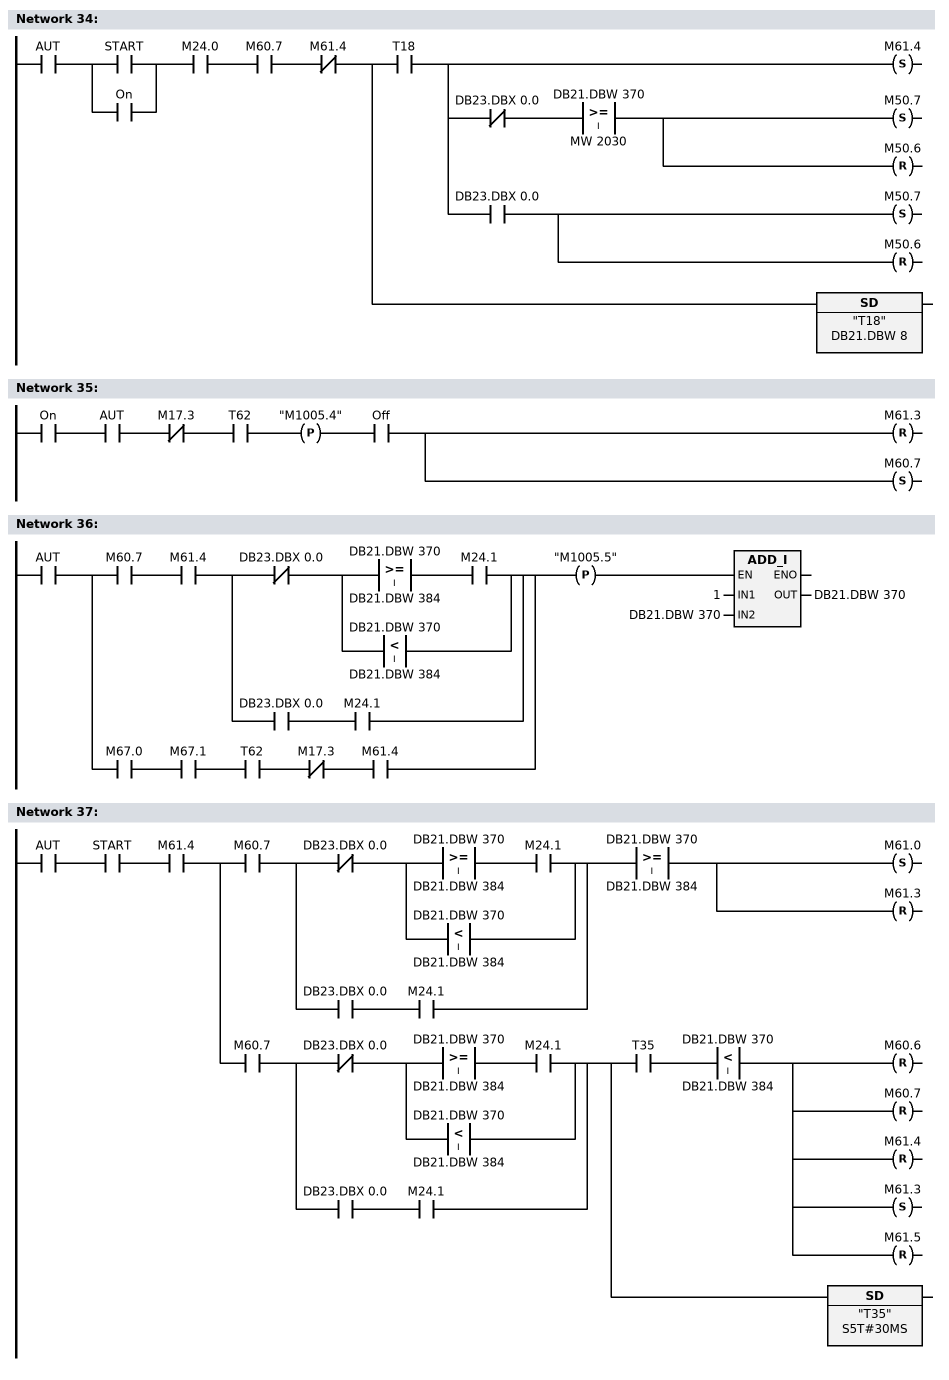
[picture p24: FC14 - AUTOMATIC networks 34-37]
NETWORK
TITLE =
      A     "AUT";
      A(;
      O     "START";
      O     "On";
      );
      A     "M24.0";
      A     "M60.7";
      AN    "M61.4";
      =     L 24.0;
      A     L 24.0;
      A     "T18";
      =     L 24.1;
      A     L 24.1;
      BLD   102;
      S     "M61.4";
      A     L 24.1;
      AN    DB23.DBX 0.0;
      A(;
      L     DB21.DBW 370;
      L     MW 2030;
      >=I;
      );
      S     "M50.7";
      R     "M50.6";
      A     L 24.1;
      A     DB23.DBX 0.0;
      S     "M50.7";
      R     "M50.6";
      A     L 24.0;
      BLD   102;
      L     DB21.DBW 8;
      SD    "T18";
NETWORK
TITLE =
      A     "On";
      A     "AUT";
      AN    "M17.3";
      A     "T62";
      FP    "M1005.4";
      A     "Off";
      R     "M61.3";
      S     "M60.7";
NETWORK
TITLE =
      A     "AUT";
      A(;
      A     "M60.7";
      A     "M61.4";
      A(;
      AN    DB23.DBX 0.0;
      A(;
      A(;
      L     DB21.DBW 370;
      L     DB21.DBW 384;
      >=I;
      );
      A     "M24.1";
      O(;
      L     DB21.DBW 370;
      L     DB21.DBW 384;
      <I;
      );
      );
      O;
      A     DB23.DBX 0.0;
      A     "M24.1";
      );
      O;
      A     "M67.0";
      A     "M67.1";
      A     "T62";
      AN    "M17.3";
      A     "M61.4";
      );
      FP    "M1005.5";
      JNB   M025;
      L     1;
      L     DB21.DBW 370;
      +I;
      T     DB21.DBW 370;
M025: NOP   0;
NETWORK
TITLE =
      A     "AUT";
      A     "START";
      A     "M61.4";
      =     L 24.0;
      A     L 24.0;
      A     "M60.7";
      A(;
      AN    DB23.DBX 0.0;
      A(;
      A(;
      L     DB21.DBW 370;
      L     DB21.DBW 384;
      >=I;
      );
      A     "M24.1";
      O(;
      L     DB21.DBW 370;
      L     DB21.DBW 384;
      <I;
      );
      );
      O;
      A     DB23.DBX 0.0;
      A     "M24.1";
      );
      A(;
      L     DB21.DBW 370;
      L     DB21.DBW 384;
      >=I;
      );
      S     "M61.0";
      R     "M61.3";
      A     L 24.0;
      A     "M60.7";
      A(;
      AN    DB23.DBX 0.0;
      A(;
      A(;
      L     DB21.DBW 370;
      L     DB21.DBW 384;
      >=I;
      );
      A     "M24.1";
      O(;
      L     DB21.DBW 370;
      L     DB21.DBW 384;
      <I;
      );
      );
      O;
      A     DB23.DBX 0.0;
      A     "M24.1";
      );
      =     L 24.1;
      A     L 24.1;
      A     "T35";
      A(;
      L     DB21.DBW 370;
      L     DB21.DBW 384;
      <I;
      );
      R     "M60.6";
      R     "M60.7";
      R     "M61.4";
      S     "M61.3";
      R     "M61.5";
      A     L 24.1;
      BLD   102;
      L     S5T#30MS;
      SD    "T35";
NETWORK
TITLE =
NETWORK
TITLE =
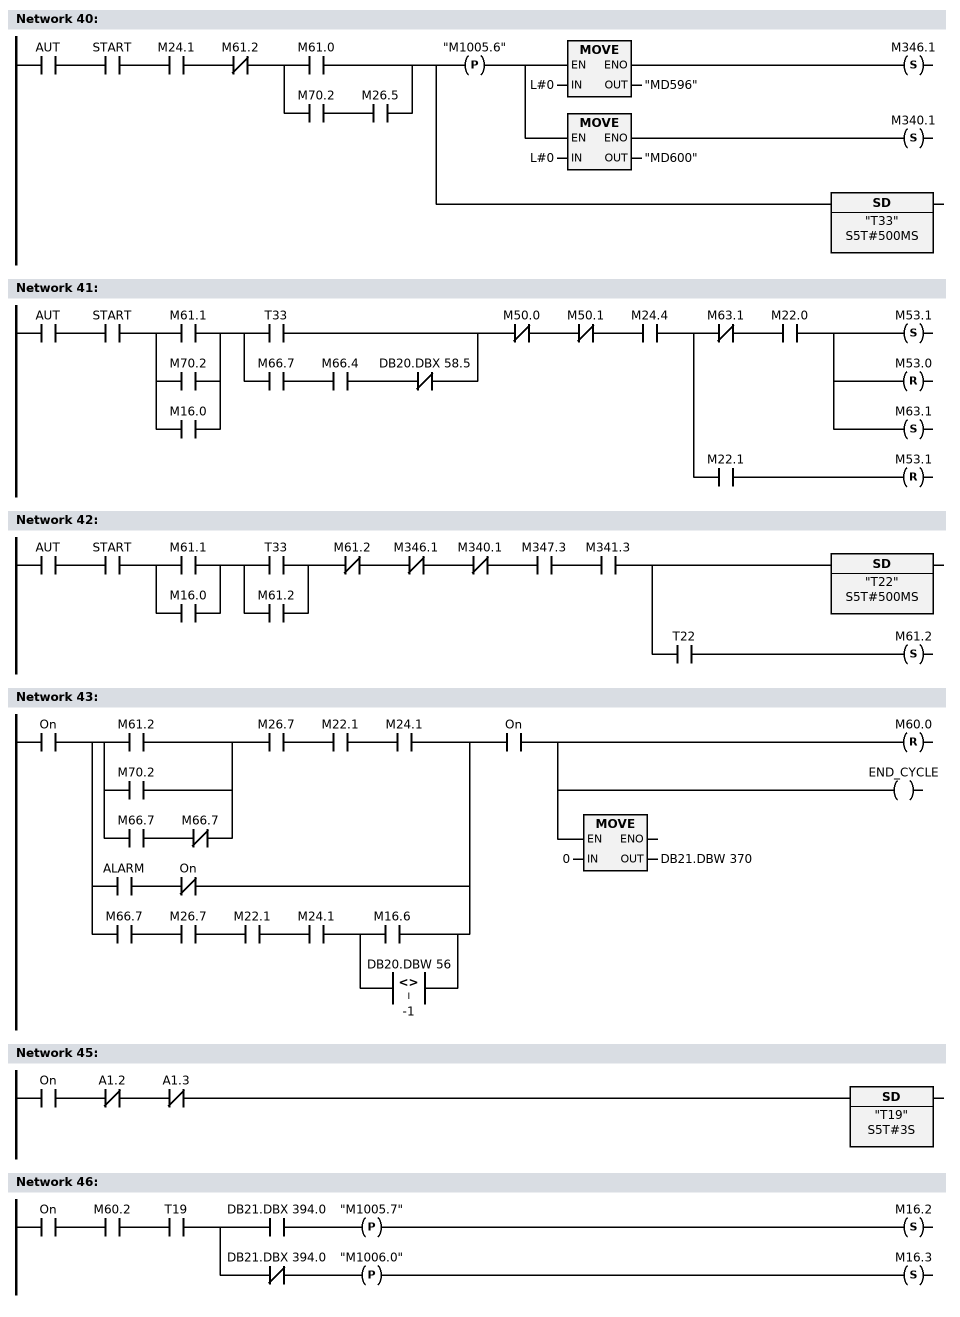
NETWORK
TITLE =
      A     "AUT";
      A     "START";
      A     "M24.1";
      AN    "M61.2";
      A(;
      O     "M61.0";
      O;
      A     "M70.2";
      A     "M26.5";
      );
      =     L 24.0;
      A     L 24.0;
      FP    "M1005.6";
      =     L 24.1;
      A     L 24.1;
      JNB   M026;
      L     L#0;
      T     "MD596";
      SET;
      SAVE;
      CLR;
M026: A     BR;
      S     "M346.1";
      A     L 24.1;
      JNB   M027;
      L     L#0;
      T     "MD600";
      SET;
      SAVE;
      CLR;
M027: A     BR;
      S     "M340.1";
      A     L 24.0;
      BLD   102;
      L     S5T#500MS;
      SD    "T33";
NETWORK
TITLE =
      A     "AUT";
      A     "START";
      A(;
      O     "M61.1";
      O     "M70.2";
      O     "M16.0";
      );
      A(;
      O     "T33";
      O;
      A     "M66.7";
      A     "M66.4";
      AN    DB20.DBX 58.5;
      );
      AN    "M50.0";
      AN    "M50.1";
      A     "M24.4";
      =     L 24.0;
      A     L 24.0;
      AN    "M63.1";
      A     "M22.0";
      S     "M53.1";
      R     "M53.0";
      S     "M63.1";
      A     L 24.0;
      A     "M22.1";
      R     "M53.1";
NETWORK
TITLE =
      A     "AUT";
      A     "START";
      A(;
      O     "M61.1";
      O     "M16.0";
      );
      A(;
      O     "T33";
      O     "M61.2";
      );
      AN    "M61.2";
      AN    "M346.1";
      AN    "M340.1";
      A     "M347.3";
      A     "M341.3";
      =     L 24.0;
      A     L 24.0;
      BLD   102;
      L     S5T#500MS;
      SD    "T22";
      A     L 24.0;
      A     "T22";
      S     "M61.2";
NETWORK
TITLE =
      A     "On";
      A(;
      A(;
      O     "M61.2";
      O     "M70.2";
      O;
      A     "M66.7";
      AN    "M66.7";
      );
      A     "M26.7";
      A     "M22.1";
      A     "M24.1";
      O;
      A     "ALARM";
      AN    "On";
      O;
      A     "M66.7";
      A     "M26.7";
      A     "M22.1";
      A     "M24.1";
      A(;
      O     "M16.6";
      O(;
      L     DB20.DBW 56;
      L     -1;
      <>I;
      );
      );
      );
      A     "On";
      =     L 24.0;
      A     L 24.0;
      BLD   102;
      R     "M60.0";
      A     L 24.0;
      BLD   102;
      =     "END_CYCLE";
      A     L 24.0;
      JNB   M028;
      L     0;
      T     DB21.DBW 370;
M028: NOP   0;
NETWORK
TITLE =
NETWORK
TITLE =
      A     "On";
      AN    "A1.2";
      AN    "A1.3";
      L     S5T#3S;
      SD    "T19";
NETWORK
TITLE =
      A     "On";
      A     "M60.2";
      A     "T19";
      =     L 24.0;
      A     L 24.0;
      A     DB21.DBX 394.0;
      FP    "M1005.7";
      S     "M16.2";
      A     L 24.0;
      AN    DB21.DBX 394.0;
      FP    "M1006.0";
      S     "M16.3";
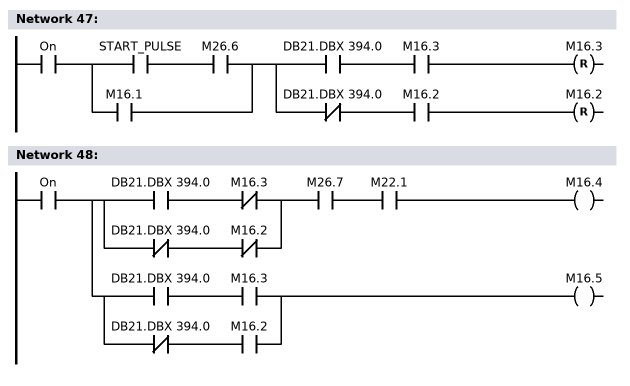
NETWORK
TITLE =
      A     "On";
      A(;
      A     "START_PULSE";
      A     "M26.6";
      O     "M16.1";
      );
      =     L 24.0;
      A     L 24.0;
      A     DB21.DBX 394.0;
      A     "M16.3";
      R     "M16.3";
      A     L 24.0;
      AN    DB21.DBX 394.0;
      A     "M16.2";
      R     "M16.2";
NETWORK
TITLE =
      A     "On";
      =     L 24.0;
      A     L 24.0;
      A(;
      A     DB21.DBX 394.0;
      AN    "M16.3";
      O;
      AN    DB21.DBX 394.0;
      AN    "M16.2";
      );
      A     "M26.7";
      A     "M22.1";
      =     "M16.4";
      A     L 24.0;
      A(;
      A     DB21.DBX 394.0;
      A     "M16.3";
      O;
      AN    DB21.DBX 394.0;
      A     "M16.2";
      );
      =     "M16.5";
END_FUNCTION

FUNCTION "FC16 - ALARMS" : VOID	// FC 16
VERSION : 0.1
BEGIN
// (block stored without names or comments; labels and parameter names are numbered)
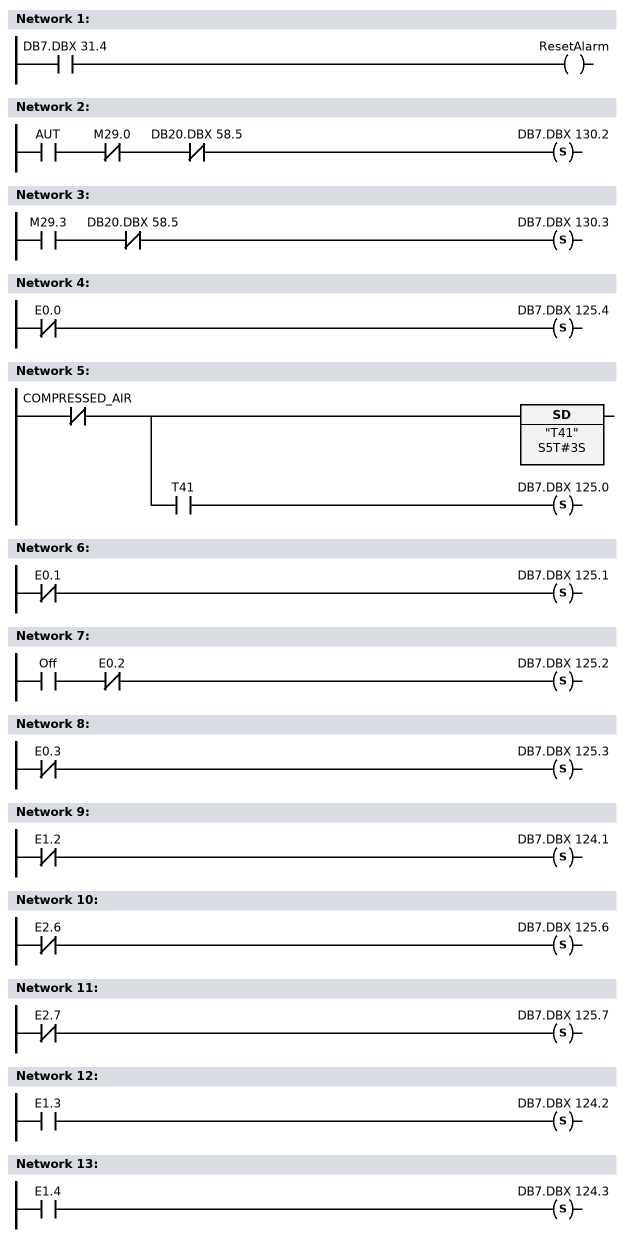
NETWORK
TITLE =
      A     DB7.DBX 31.4;
      =     "ResetAlarm";
NETWORK
TITLE =
      A     "AUT";
      AN    "M29.0";
      AN    DB20.DBX 58.5;
      S     DB7.DBX 130.2;
NETWORK
TITLE =
      A     "M29.3";
      AN    DB20.DBX 58.5;
      S     DB7.DBX 130.3;
NETWORK
TITLE =
      AN    "E0.0";
      S     DB7.DBX 125.4;
NETWORK
TITLE =
      AN    "COMPRESSED_AIR";
      =     L 1.0;
      A     L 1.0;
      BLD   102;
      L     S5T#3S;
      SD    "T41";
      A     L 1.0;
      A     "T41";
      S     DB7.DBX 125.0;
NETWORK
TITLE =
      AN    "E0.1";
      S     DB7.DBX 125.1;
NETWORK
TITLE =
      A     "Off";
      AN    "E0.2";
      S     DB7.DBX 125.2;
NETWORK
TITLE =
      AN    "E0.3";
      S     DB7.DBX 125.3;
NETWORK
TITLE =
      AN    "E1.2";
      S     DB7.DBX 124.1;
NETWORK
TITLE =
      AN    "E2.6";
      S     DB7.DBX 125.6;
NETWORK
TITLE =
      AN    "E2.7";
      S     DB7.DBX 125.7;
NETWORK
TITLE =
      A     "E1.3";
      S     DB7.DBX 124.2;
NETWORK
TITLE =
      A     "E1.4";
      S     DB7.DBX 124.3;
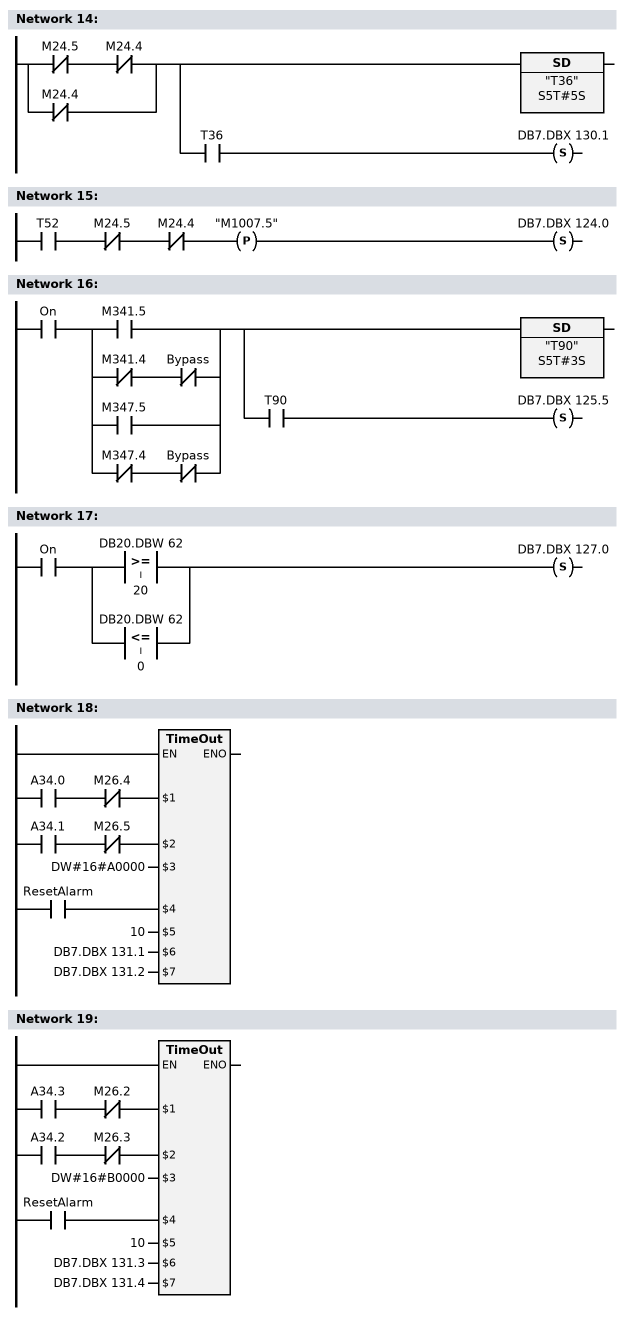
NETWORK
TITLE =
      AN    "M24.5";
      AN    "M24.4";
      ON    "M24.4";
      =     L 1.0;
      A     L 1.0;
      BLD   102;
      L     S5T#5S;
      SD    "T36";
      A     L 1.0;
      A     "T36";
      S     DB7.DBX 130.1;
NETWORK
TITLE =
      A     "T52";
      AN    "M24.5";
      AN    "M24.4";
      FP    "M1007.5";
      S     DB7.DBX 124.0;
NETWORK
TITLE =
      A     "On";
      A(;
      O     "M341.5";
      O;
      AN    "M341.4";
      AN    "Bypass";
      O     "M347.5";
      O;
      AN    "M347.4";
      AN    "Bypass";
      );
      =     L 1.0;
      A     L 1.0;
      BLD   102;
      L     S5T#3S;
      SD    "T90";
      A     L 1.0;
      A     "T90";
      S     DB7.DBX 125.5;
NETWORK
TITLE =
      A     "On";
      A(;
      O(;
      L     DB20.DBW 62;
      L     20;
      >=I;
      );
      O(;
      L     DB20.DBW 62;
      L     0;
      <=I;
      );
      );
      S     DB7.DBX 127.0;
NETWORK
TITLE =
      A     "A34.0";
      AN    "M26.4";
      =     L 1.0;
      BLD   103;
      A     "A34.1";
      AN    "M26.5";
      =     L 1.1;
      BLD   103;
      A     "ResetAlarm";
      =     L 1.2;
      BLD   103;
      CALL  "TimeOut" (
           $1                       := L 1.0,
           $2                       := L 1.1,
           $3                       := DW#16#A0000,
           $4                       := L 1.2,
           $5                       := 10,
           $6                       := DB7.DBX 131.1,
           $7                       := DB7.DBX 131.2);
      NOP   0;
NETWORK
TITLE =
      A     "A34.3";
      AN    "M26.2";
      =     L 1.0;
      BLD   103;
      A     "A34.2";
      AN    "M26.3";
      =     L 1.1;
      BLD   103;
      A     "ResetAlarm";
      =     L 1.2;
      BLD   103;
      CALL  "TimeOut" (
           $1                       := L 1.0,
           $2                       := L 1.1,
           $3                       := DW#16#B0000,
           $4                       := L 1.2,
           $5                       := 10,
           $6                       := DB7.DBX 131.3,
           $7                       := DB7.DBX 131.4);
      NOP   0;
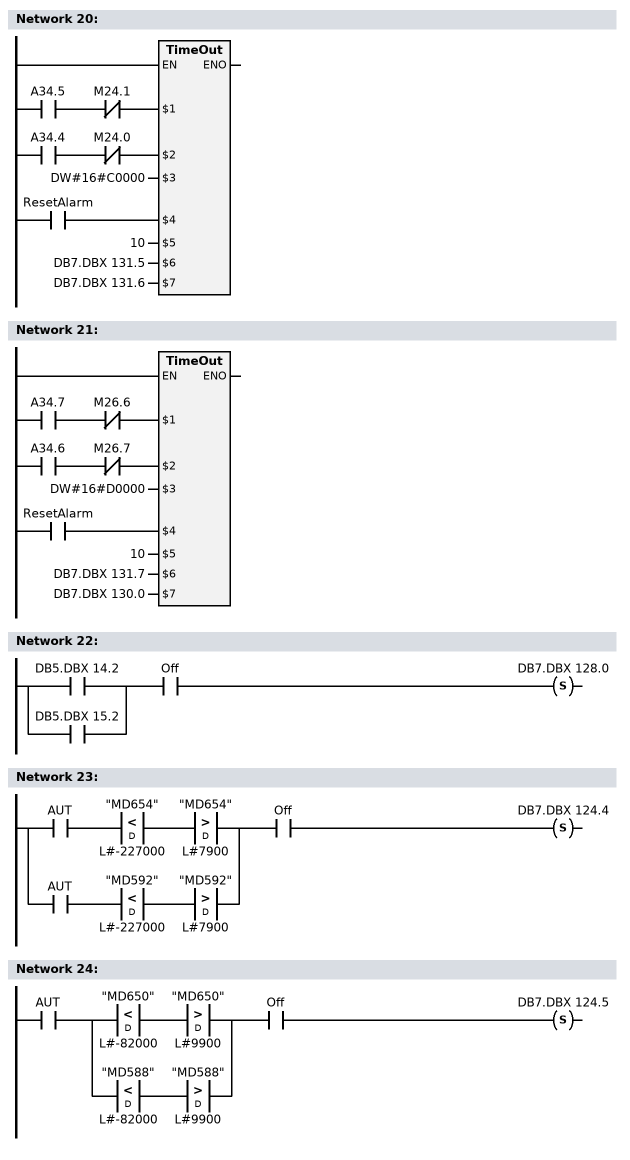
NETWORK
TITLE =
      A     "A34.5";
      AN    "M24.1";
      =     L 1.0;
      BLD   103;
      A     "A34.4";
      AN    "M24.0";
      =     L 1.1;
      BLD   103;
      A     "ResetAlarm";
      =     L 1.2;
      BLD   103;
      CALL  "TimeOut" (
           $1                       := L 1.0,
           $2                       := L 1.1,
           $3                       := DW#16#C0000,
           $4                       := L 1.2,
           $5                       := 10,
           $6                       := DB7.DBX 131.5,
           $7                       := DB7.DBX 131.6);
      NOP   0;
NETWORK
TITLE =
      A     "A34.7";
      AN    "M26.6";
      =     L 1.0;
      BLD   103;
      A     "A34.6";
      AN    "M26.7";
      =     L 1.1;
      BLD   103;
      A     "ResetAlarm";
      =     L 1.2;
      BLD   103;
      CALL  "TimeOut" (
           $1                       := L 1.0,
           $2                       := L 1.1,
           $3                       := DW#16#D0000,
           $4                       := L 1.2,
           $5                       := 10,
           $6                       := DB7.DBX 131.7,
           $7                       := DB7.DBX 130.0);
      NOP   0;
NETWORK
TITLE =
      A(;
      O     DB5.DBX 14.2;
      O     DB5.DBX 15.2;
      );
      A     "Off";
      S     DB7.DBX 128.0;
NETWORK
TITLE =
      A(;
      A     "AUT";
      A(;
      L     "MD654";
      L     L#-227000;
      <D;
      );
      A(;
      L     "MD654";
      L     L#7900;
      >D;
      );
      O;
      A     "AUT";
      A(;
      L     "MD592";
      L     L#-227000;
      <D;
      );
      A(;
      L     "MD592";
      L     L#7900;
      >D;
      );
      );
      A     "Off";
      S     DB7.DBX 124.4;
NETWORK
TITLE =
      A     "AUT";
      A(;
      A(;
      L     "MD650";
      L     L#-82000;
      <D;
      );
      A(;
      L     "MD650";
      L     L#9900;
      >D;
      );
      O;
      A(;
      L     "MD588";
      L     L#-82000;
      <D;
      );
      A(;
      L     "MD588";
      L     L#9900;
      >D;
      );
      );
      A     "Off";
      S     DB7.DBX 124.5;
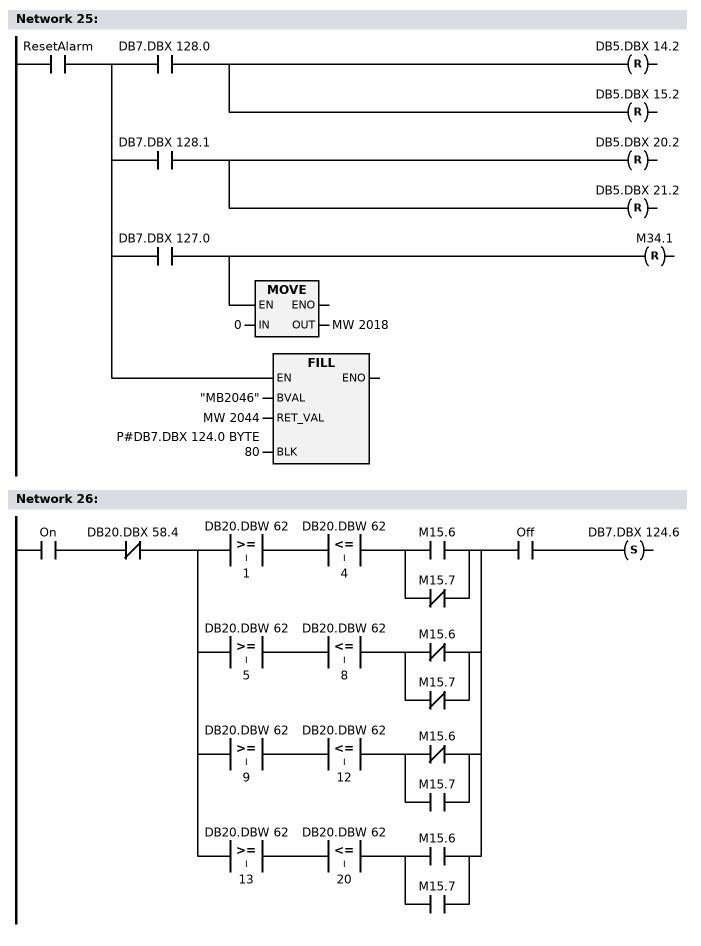
NETWORK
TITLE =
      A     "ResetAlarm";
      =     L 1.0;
      A     L 1.0;
      A     DB7.DBX 128.0;
      R     DB5.DBX 14.2;
      R     DB5.DBX 15.2;
      A     L 1.0;
      A     DB7.DBX 128.1;
      R     DB5.DBX 20.2;
      R     DB5.DBX 21.2;
      A     L 1.0;
      A     DB7.DBX 127.0;
      =     L 1.1;
      A     L 1.1;
      BLD   102;
      R     "M34.1";
      A     L 1.1;
      JNB   M001;
      L     0;
      T     MW 2018;
M001: NOP   0;
      A     L 1.0;
      JNB   M002;
      CALL  "FILL" (
           BVAL                     := "MB2046",
           RET_VAL                  := MW 2044,
           BLK                      := P#DB7.DBX 124.0 BYTE 80);
M002: NOP   0;
NETWORK
TITLE =
      A     "On";
      AN    DB20.DBX 58.4;
      A(;
      A(;
      L     DB20.DBW 62;
      L     1;
      >=I;
      );
      A(;
      L     DB20.DBW 62;
      L     4;
      <=I;
      );
      A(;
      O     "M15.6";
      ON    "M15.7";
      );
      O;
      A(;
      L     DB20.DBW 62;
      L     5;
      >=I;
      );
      A(;
      L     DB20.DBW 62;
      L     8;
      <=I;
      );
      A(;
      ON    "M15.6";
      ON    "M15.7";
      );
      O;
      A(;
      L     DB20.DBW 62;
      L     9;
      >=I;
      );
      A(;
      L     DB20.DBW 62;
      L     12;
      <=I;
      );
      A(;
      ON    "M15.6";
      O     "M15.7";
      );
      O;
      A(;
      L     DB20.DBW 62;
      L     13;
      >=I;
      );
      A(;
      L     DB20.DBW 62;
      L     20;
      <=I;
      );
      A(;
      O     "M15.6";
      O     "M15.7";
      );
      );
      A     "Off";
      S     DB7.DBX 124.6;
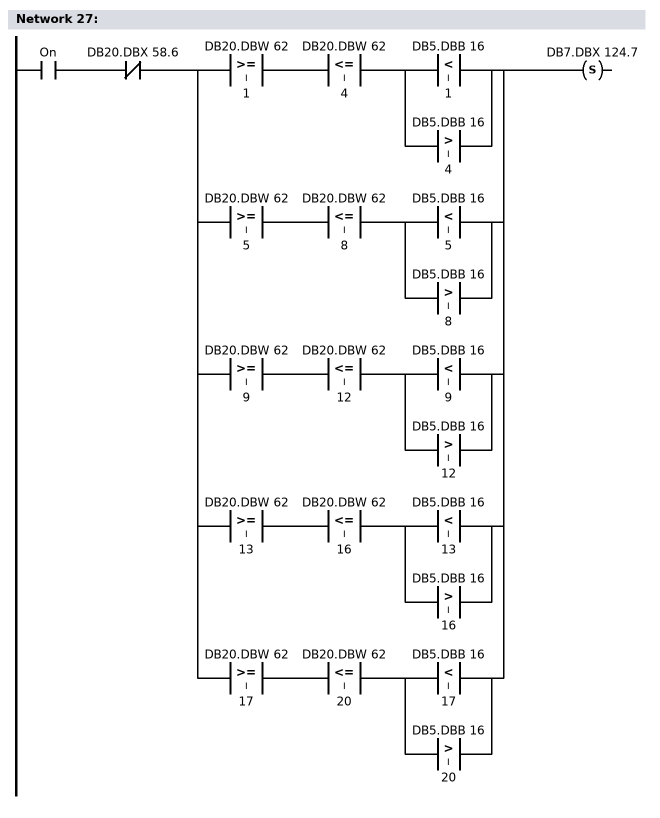
NETWORK
TITLE =
      A     "On";
      AN    DB20.DBX 58.6;
      A(;
      A(;
      L     DB20.DBW 62;
      L     1;
      >=I;
      );
      A(;
      L     DB20.DBW 62;
      L     4;
      <=I;
      );
      A(;
      O(;
      L     DB5.DBB 16;
      L     1;
      <I;
      );
      O(;
      L     DB5.DBB 16;
      L     4;
      >I;
      );
      );
      O;
      A(;
      L     DB20.DBW 62;
      L     5;
      >=I;
      );
      A(;
      L     DB20.DBW 62;
      L     8;
      <=I;
      );
      A(;
      O(;
      L     DB5.DBB 16;
      L     5;
      <I;
      );
      O(;
      L     DB5.DBB 16;
      L     8;
      >I;
      );
      );
      O;
      A(;
      L     DB20.DBW 62;
      L     9;
      >=I;
      );
      A(;
      L     DB20.DBW 62;
      L     12;
      <=I;
      );
      A(;
      O(;
      L     DB5.DBB 16;
      L     9;
      <I;
      );
      O(;
      L     DB5.DBB 16;
      L     12;
      >I;
      );
      );
      O;
      A(;
      L     DB20.DBW 62;
      L     13;
      >=I;
      );
      A(;
      L     DB20.DBW 62;
      L     16;
      <=I;
      );
      A(;
      O(;
      L     DB5.DBB 16;
      L     13;
      <I;
      );
      O(;
      L     DB5.DBB 16;
      L     16;
      >I;
      );
      );
      O;
      A(;
      L     DB20.DBW 62;
      L     17;
      >=I;
      );
      A(;
      L     DB20.DBW 62;
      L     20;
      <=I;
      );
      A(;
      O(;
      L     DB5.DBB 16;
      L     17;
      <I;
      );
      O(;
      L     DB5.DBB 16;
      L     20;
      >I;
      );
      );
      );
      S     DB7.DBX 124.7;
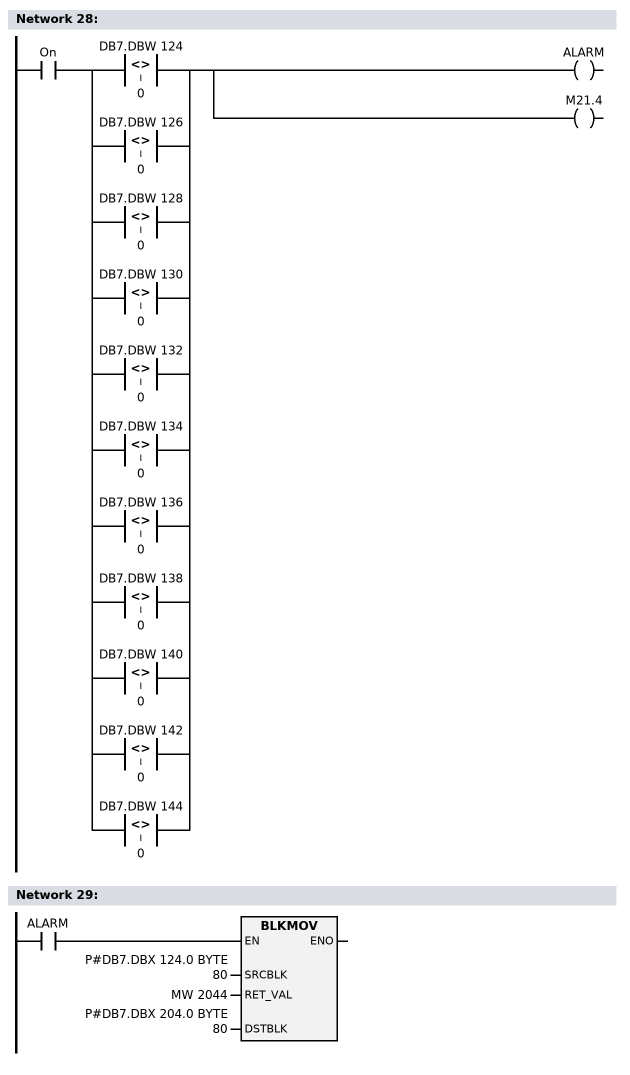
NETWORK
TITLE =
      A     "On";
      A(;
      O(;
      L     DB7.DBW 124;
      L     0;
      <>I;
      );
      O(;
      L     DB7.DBW 126;
      L     0;
      <>I;
      );
      O(;
      L     DB7.DBW 128;
      L     0;
      <>I;
      );
      O(;
      L     DB7.DBW 130;
      L     0;
      <>I;
      );
      O(;
      L     DB7.DBW 132;
      L     0;
      <>I;
      );
      O(;
      L     DB7.DBW 134;
      L     0;
      <>I;
      );
      O(;
      L     DB7.DBW 136;
      L     0;
      <>I;
      );
      O(;
      L     DB7.DBW 138;
      L     0;
      <>I;
      );
      O(;
      L     DB7.DBW 140;
      L     0;
      <>I;
      );
      O(;
      L     DB7.DBW 142;
      L     0;
      <>I;
      );
      O(;
      L     DB7.DBW 144;
      L     0;
      <>I;
      );
      );
      =     "ALARM";
      =     "M21.4";
NETWORK
TITLE =
      A     "ALARM";
      JNB   M003;
      CALL  "BLKMOV" (
           SRCBLK                   := P#DB7.DBX 124.0 BYTE 80,
           RET_VAL                  := MW 2044,
           DSTBLK                   := P#DB7.DBX 204.0 BYTE 80);
M003: NOP   0;
END_FUNCTION

FUNCTION "FC17 - OPERATOR PANNEL" : VOID	// FC 17
VERSION : 0.1
BEGIN
// (block stored without names or comments; labels and parameter names are numbered)
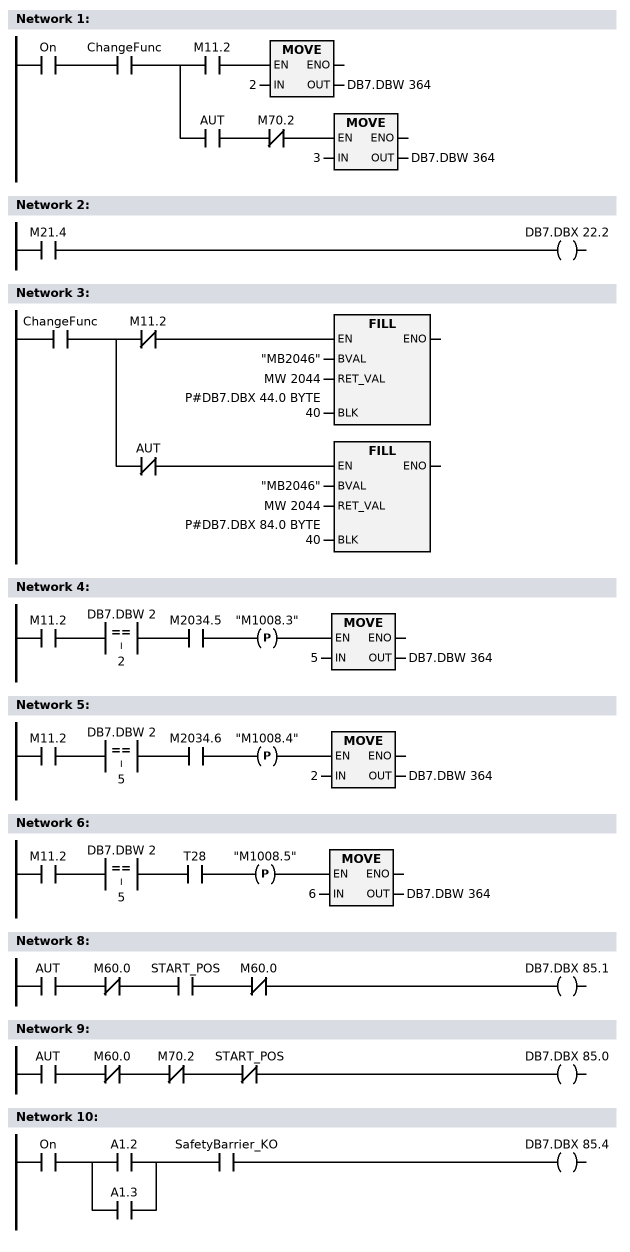
NETWORK
TITLE =
      A     "On";
      A     "ChangeFunc";
      =     L 0.0;
      A     L 0.0;
      A     "M11.2";
      JNB   M001;
      L     2;
      T     DB7.DBW 364;
M001: NOP   0;
      A     L 0.0;
      A     "AUT";
      AN    "M70.2";
      JNB   M002;
      L     3;
      T     DB7.DBW 364;
M002: NOP   0;
NETWORK
TITLE =
      A     "M21.4";
      =     DB7.DBX 22.2;
NETWORK
TITLE =
      A     "ChangeFunc";
      =     L 0.0;
      A     L 0.0;
      AN    "M11.2";
      JNB   M003;
      CALL  "FILL" (
           BVAL                     := "MB2046",
           RET_VAL                  := MW 2044,
           BLK                      := P#DB7.DBX 44.0 BYTE 40);
M003: NOP   0;
      A     L 0.0;
      AN    "AUT";
      JNB   M004;
      CALL  "FILL" (
           BVAL                     := "MB2046",
           RET_VAL                  := MW 2044,
           BLK                      := P#DB7.DBX 84.0 BYTE 40);
M004: NOP   0;
NETWORK
TITLE =
      A     "M11.2";
      A(;
      L     DB7.DBW 2;
      L     2;
      ==I;
      );
      A     "M2034.5";
      FP    "M1008.3";
      JNB   M005;
      L     5;
      T     DB7.DBW 364;
M005: NOP   0;
NETWORK
TITLE =
      A     "M11.2";
      A(;
      L     DB7.DBW 2;
      L     5;
      ==I;
      );
      A     "M2034.6";
      FP    "M1008.4";
      JNB   M006;
      L     2;
      T     DB7.DBW 364;
M006: NOP   0;
NETWORK
TITLE =
      A     "M11.2";
      A(;
      L     DB7.DBW 2;
      L     5;
      ==I;
      );
      A     "T28";
      FP    "M1008.5";
      JNB   M007;
      L     6;
      T     DB7.DBW 364;
M007: NOP   0;
NETWORK
TITLE =
NETWORK
TITLE =
      A     "AUT";
      AN    "M60.0";
      A     "START_POS";
      AN    "M60.0";
      =     DB7.DBX 85.1;
NETWORK
TITLE =
      A     "AUT";
      AN    "M60.0";
      AN    "M70.2";
      AN    "START_POS";
      =     DB7.DBX 85.0;
NETWORK
TITLE =
      A     "On";
      A(;
      O     "A1.2";
      O     "A1.3";
      );
      A     "SafetyBarrier_KO";
      =     DB7.DBX 85.4;
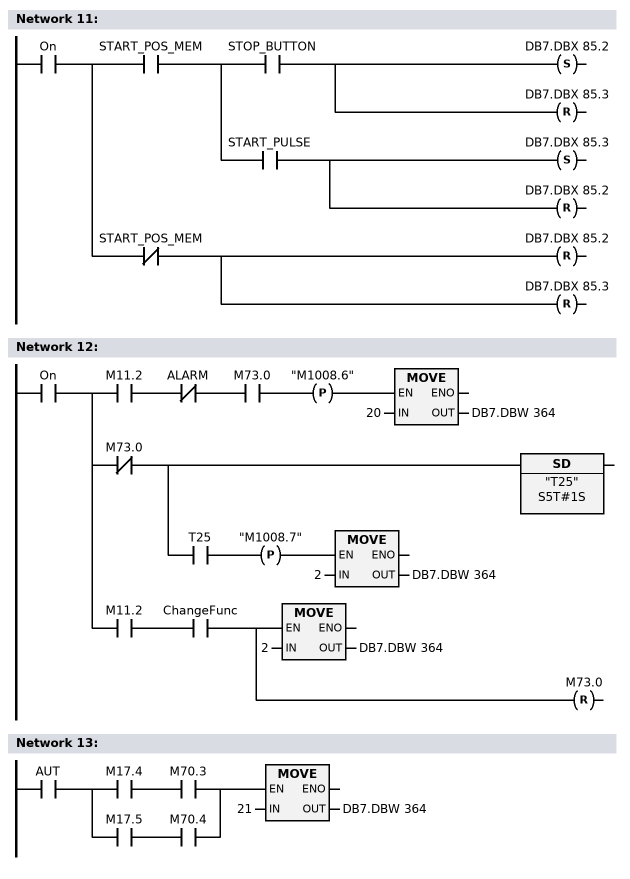
NETWORK
TITLE =
      A     "On";
      =     L 0.0;
      A     L 0.0;
      A     "START_POS_MEM";
      =     L 0.1;
      A     L 0.1;
      A     "STOP_BUTTON";
      S     DB7.DBX 85.2;
      R     DB7.DBX 85.3;
      A     L 0.1;
      A     "START_PULSE";
      S     DB7.DBX 85.3;
      R     DB7.DBX 85.2;
      A     L 0.0;
      AN    "START_POS_MEM";
      R     DB7.DBX 85.2;
      R     DB7.DBX 85.3;
NETWORK
TITLE =
      A     "On";
      =     L 0.0;
      A     L 0.0;
      A     "M11.2";
      AN    "ALARM";
      A     "M73.0";
      FP    "M1008.6";
      JNB   M008;
      L     20;
      T     DB7.DBW 364;
M008: NOP   0;
      A     L 0.0;
      AN    "M73.0";
      =     L 0.1;
      A     L 0.1;
      BLD   102;
      L     S5T#1S;
      SD    "T25";
      A     L 0.1;
      A     "T25";
      FP    "M1008.7";
      JNB   M009;
      L     2;
      T     DB7.DBW 364;
M009: NOP   0;
      A     L 0.0;
      A     "M11.2";
      A     "ChangeFunc";
      =     L 0.1;
      A     L 0.1;
      JNB   M010;
      L     2;
      T     DB7.DBW 364;
M010: NOP   0;
      A     L 0.1;
      BLD   102;
      R     "M73.0";
NETWORK
TITLE =
      A     "AUT";
      A(;
      A     "M17.4";
      A     "M70.3";
      O;
      A     "M17.5";
      A     "M70.4";
      );
      JNB   M011;
      L     21;
      T     DB7.DBW 364;
M011: NOP   0;
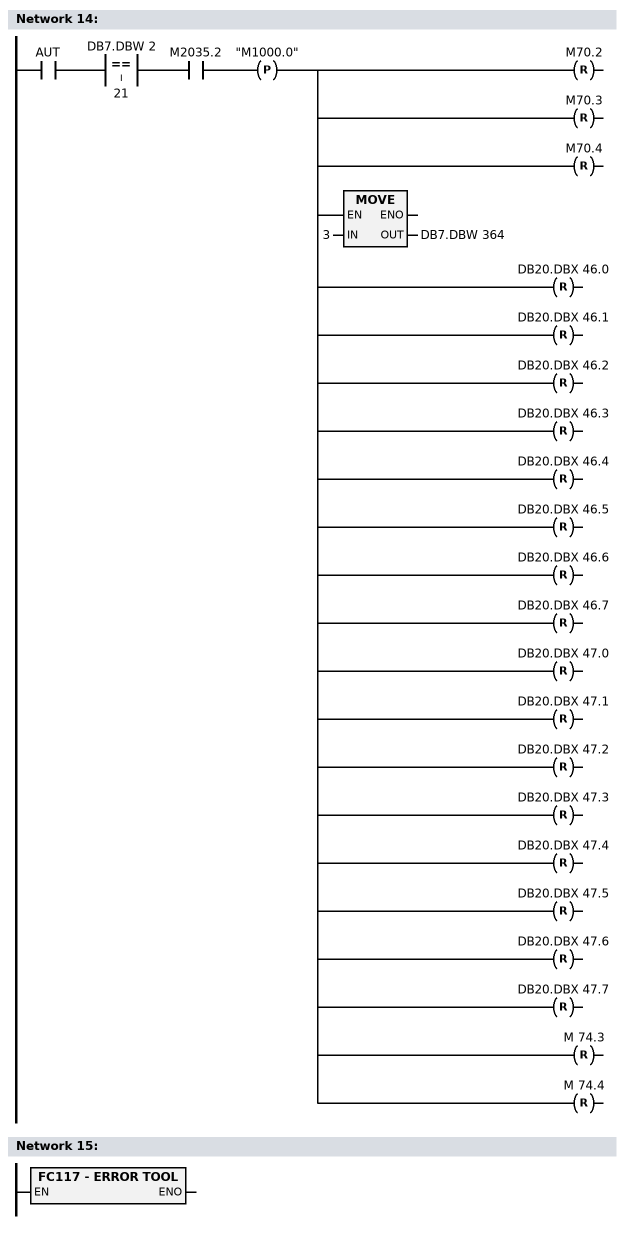
NETWORK
TITLE =
      A     "AUT";
      A(;
      L     DB7.DBW 2;
      L     21;
      ==I;
      );
      A     "M2035.2";
      FP    "M1000.0";
      =     L 0.0;
      A     L 0.0;
      BLD   102;
      R     "M70.2";
      A     L 0.0;
      BLD   102;
      R     "M70.3";
      A     L 0.0;
      BLD   102;
      R     "M70.4";
      A     L 0.0;
      JNB   M012;
      L     3;
      T     DB7.DBW 364;
M012: NOP   0;
      A     L 0.0;
      BLD   102;
      R     DB20.DBX 46.0;
      A     L 0.0;
      BLD   102;
      R     DB20.DBX 46.1;
      A     L 0.0;
      BLD   102;
      R     DB20.DBX 46.2;
      A     L 0.0;
      BLD   102;
      R     DB20.DBX 46.3;
      A     L 0.0;
      BLD   102;
      R     DB20.DBX 46.4;
      A     L 0.0;
      BLD   102;
      R     DB20.DBX 46.5;
      A     L 0.0;
      BLD   102;
      R     DB20.DBX 46.6;
      A     L 0.0;
      BLD   102;
      R     DB20.DBX 46.7;
      A     L 0.0;
      BLD   102;
      R     DB20.DBX 47.0;
      A     L 0.0;
      BLD   102;
      R     DB20.DBX 47.1;
      A     L 0.0;
      BLD   102;
      R     DB20.DBX 47.2;
      A     L 0.0;
      BLD   102;
      R     DB20.DBX 47.3;
      A     L 0.0;
      BLD   102;
      R     DB20.DBX 47.4;
      A     L 0.0;
      BLD   102;
      R     DB20.DBX 47.5;
      A     L 0.0;
      BLD   102;
      R     DB20.DBX 47.6;
      A     L 0.0;
      BLD   102;
      R     DB20.DBX 47.7;
      A     L 0.0;
      BLD   102;
      R     M 74.3;
      A     L 0.0;
      BLD   102;
      R     M 74.4;
NETWORK
TITLE =
      CALL  "FC117 - ERROR TOOL";
      NOP   0;
END_FUNCTION

FUNCTION "FC18 - OUTPUTS" : VOID	// FC 18
VERSION : 0.1
BEGIN
// (block stored without names or comments; labels and parameter names are numbered)
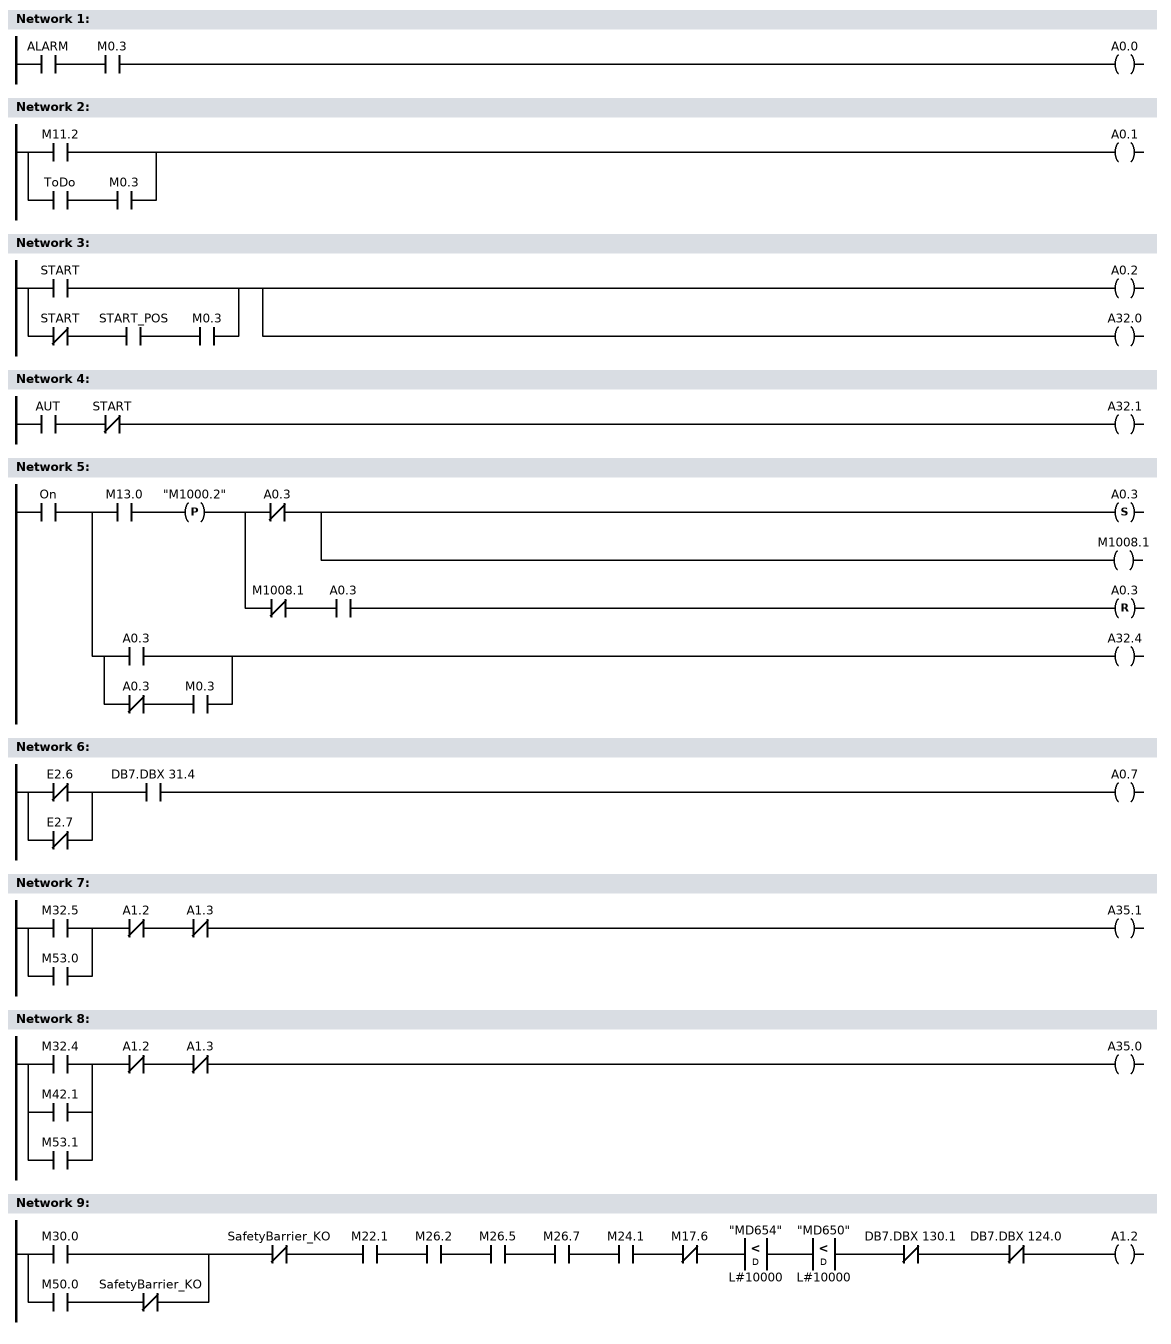
NETWORK
TITLE =
      A     "ALARM";
      A     "M0.3";
      =     "A0.0";
NETWORK
TITLE =
      O     "M11.2";
      O;
      A     "ToDo";
      A     "M0.3";
      =     "A0.1";
NETWORK
TITLE =
      O     "START";
      O;
      AN    "START";
      A     "START_POS";
      A     "M0.3";
      =     "A0.2";
      =     "A32.0";
NETWORK
TITLE =
      A     "AUT";
      AN    "START";
      =     "A32.1";
NETWORK
TITLE =
      A     "On";
      =     L 0.0;
      A     L 0.0;
      A     "M13.0";
      FP    "M1000.2";
      =     L 0.1;
      A     L 0.1;
      AN    "A0.3";
      S     "A0.3";
      =     "M1008.1";
      A     L 0.1;
      AN    "M1008.1";
      A     "A0.3";
      R     "A0.3";
      A     L 0.0;
      A(;
      O     "A0.3";
      O;
      AN    "A0.3";
      A     "M0.3";
      );
      =     "A32.4";
NETWORK
TITLE =
      A(;
      ON    "E2.6";
      ON    "E2.7";
      );
      A     DB7.DBX 31.4;
      =     "A0.7";
NETWORK
TITLE =
      A(;
      O     "M32.5";
      O     "M53.0";
      );
      AN    "A1.2";
      AN    "A1.3";
      =     "A35.1";
NETWORK
TITLE =
      A(;
      O     "M32.4";
      O     "M42.1";
      O     "M53.1";
      );
      AN    "A1.2";
      AN    "A1.3";
      =     "A35.0";
NETWORK
TITLE =
      A(;
      O     "M30.0";
      O;
      A     "M50.0";
      AN    "SafetyBarrier_KO";
      );
      AN    "SafetyBarrier_KO";
      A     "M22.1";
      A     "M26.2";
      A     "M26.5";
      A     "M26.7";
      A     "M24.1";
      AN    "M17.6";
      A(;
      L     "MD654";
      L     L#10000;
      <D;
      );
      A(;
      L     "MD650";
      L     L#10000;
      <D;
      );
      AN    DB7.DBX 130.1;
      AN    DB7.DBX 124.0;
      =     "A1.2";
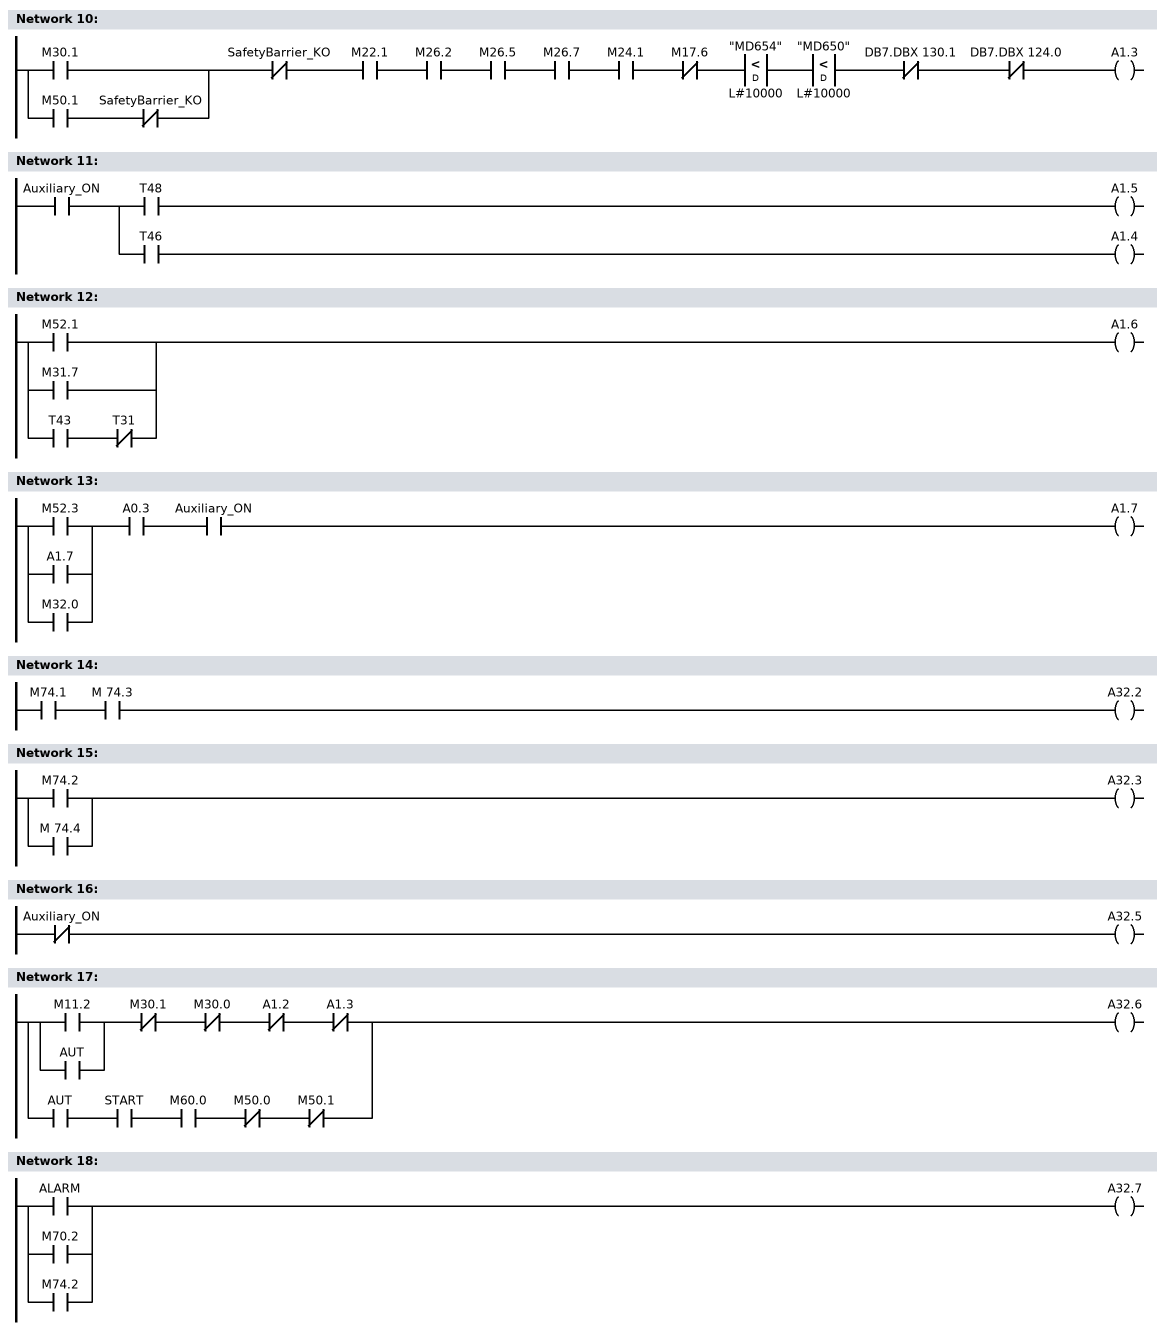
NETWORK
TITLE =
      A(;
      O     "M30.1";
      O;
      A     "M50.1";
      AN    "SafetyBarrier_KO";
      );
      AN    "SafetyBarrier_KO";
      A     "M22.1";
      A     "M26.2";
      A     "M26.5";
      A     "M26.7";
      A     "M24.1";
      AN    "M17.6";
      A(;
      L     "MD654";
      L     L#10000;
      <D;
      );
      A(;
      L     "MD650";
      L     L#10000;
      <D;
      );
      AN    DB7.DBX 130.1;
      AN    DB7.DBX 124.0;
      =     "A1.3";
NETWORK
TITLE =
      A     "Auxiliary_ON";
      =     L 0.0;
      A     L 0.0;
      A     "T48";
      =     "A1.5";
      A     L 0.0;
      A     "T46";
      =     "A1.4";
NETWORK
TITLE =
      O     "M52.1";
      O     "M31.7";
      O;
      A     "T43";
      AN    "T31";
      =     "A1.6";
NETWORK
TITLE =
      A(;
      O     "M52.3";
      O     "A1.7";
      O     "M32.0";
      );
      A     "A0.3";
      A     "Auxiliary_ON";
      =     "A1.7";
NETWORK
TITLE =
      A     "M74.1";
      A     M 74.3;
      =     "A32.2";
NETWORK
TITLE =
      O     "M74.2";
      O     M 74.4;
      =     "A32.3";
NETWORK
TITLE =
      AN    "Auxiliary_ON";
      =     "A32.5";
NETWORK
TITLE =
      A(;
      O     "M11.2";
      O     "AUT";
      );
      AN    "M30.1";
      AN    "M30.0";
      AN    "A1.2";
      AN    "A1.3";
      O;
      A     "AUT";
      A     "START";
      A     "M60.0";
      AN    "M50.0";
      AN    "M50.1";
      =     "A32.6";
NETWORK
TITLE =
      O     "ALARM";
      O     "M70.2";
      O     "M74.2";
      =     "A32.7";
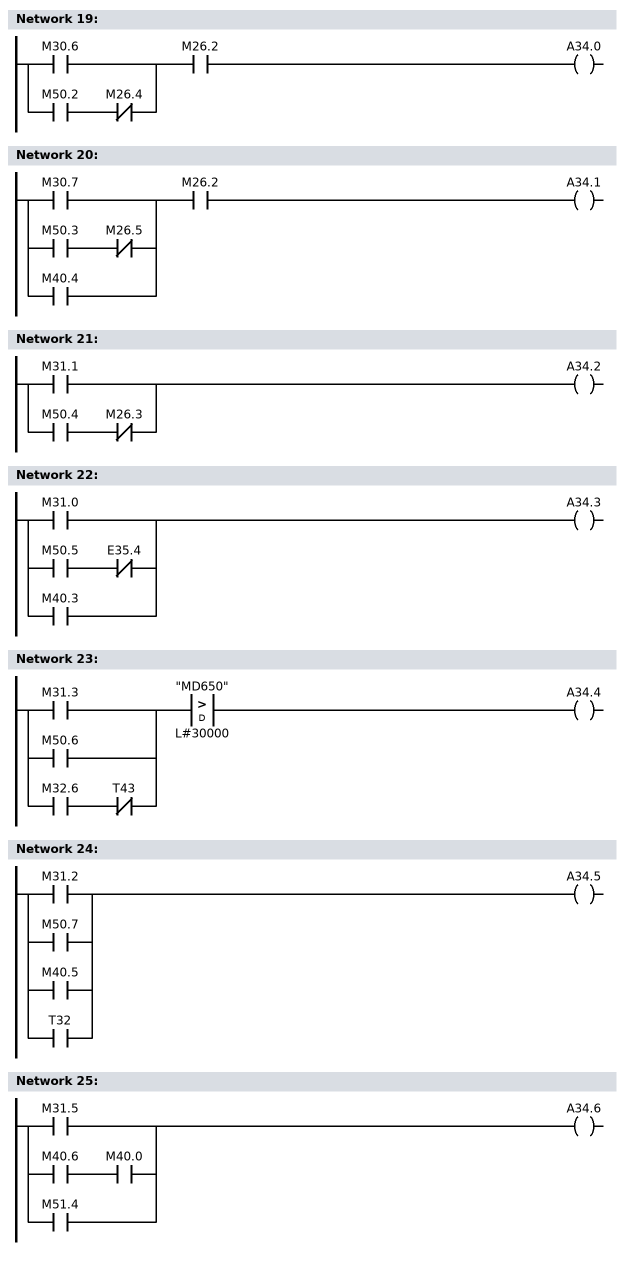
NETWORK
TITLE =
      A(;
      O     "M30.6";
      O;
      A     "M50.2";
      AN    "M26.4";
      );
      A     "M26.2";
      =     "A34.0";
NETWORK
TITLE =
      A(;
      O     "M30.7";
      O;
      A     "M50.3";
      AN    "M26.5";
      O     "M40.4";
      );
      A     "M26.2";
      =     "A34.1";
NETWORK
TITLE =
      O     "M31.1";
      O;
      A     "M50.4";
      AN    "M26.3";
      =     "A34.2";
NETWORK
TITLE =
      O     "M31.0";
      O;
      A     "M50.5";
      AN    "E35.4";
      O     "M40.3";
      =     "A34.3";
NETWORK
TITLE =
      A(;
      O     "M31.3";
      O     "M50.6";
      O;
      A     "M32.6";
      AN    "T43";
      );
      A(;
      L     "MD650";
      L     L#30000;
      >D;
      );
      =     "A34.4";
NETWORK
TITLE =
      O     "M31.2";
      O     "M50.7";
      O     "M40.5";
      O     "T32";
      =     "A34.5";
NETWORK
TITLE =
      O     "M31.5";
      O;
      A     "M40.6";
      A     "M40.0";
      O     "M51.4";
      =     "A34.6";
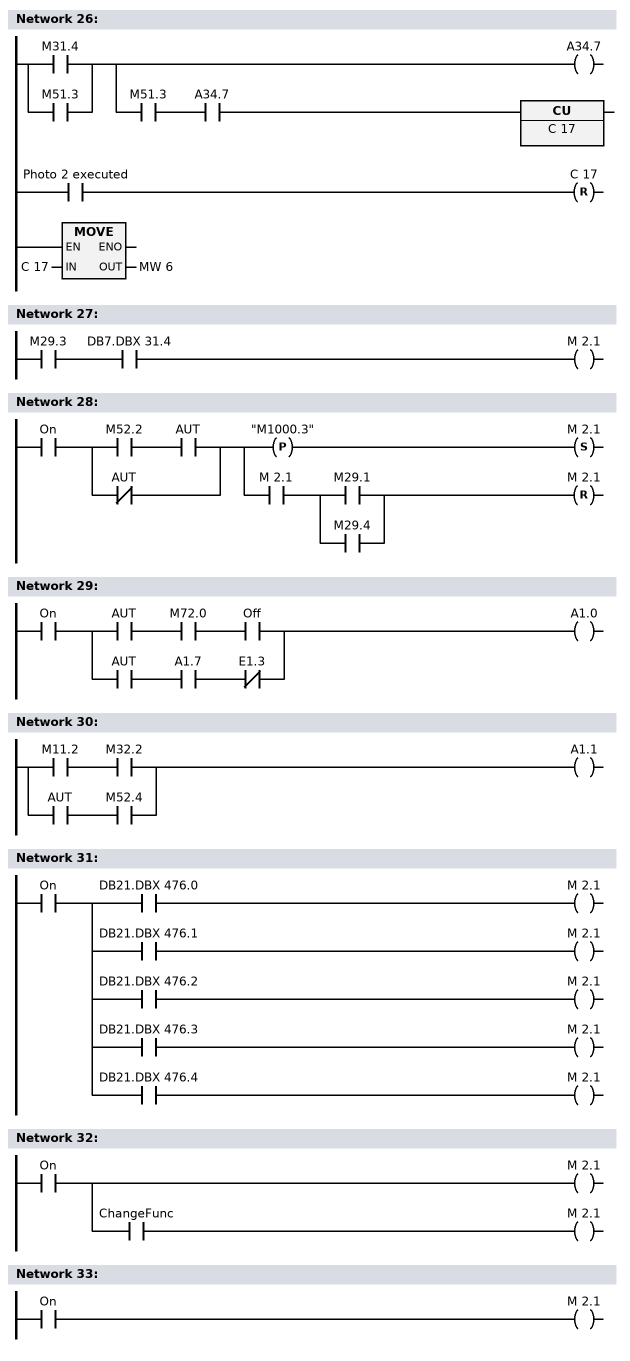
NETWORK
TITLE =
      O     "M31.4";
      O     "M51.3";
      =     L 0.0;
      A     L 0.0;
      BLD   102;
      =     "A34.7";
      A     L 0.0;
      A     "M51.3";
      A     "A34.7";
      CU    C 17;
      BLD   101;
      NOP   0;
      NOP   0;
      A     "Photo 2 executed";
      R     C 17;
      L     C 17;
      T     MW 6;
      NOP   0;
      NOP   0;
NETWORK
TITLE =
      A     "M29.3";
      A     DB7.DBX 31.4;
      =     M 2.1;
NETWORK
TITLE =
      A     "On";
      A(;
      A     "M52.2";
      A     "AUT";
      ON    "AUT";
      );
      =     L 0.0;
      A     L 0.0;
      FP    "M1000.3";
      S     M 2.1;
      A     L 0.0;
      A     M 2.1;
      A(;
      O     "M29.1";
      O     "M29.4";
      );
      R     M 2.1;
NETWORK
TITLE =
      A     "On";
      A(;
      A     "AUT";
      A     "M72.0";
      A     "Off";
      O;
      A     "AUT";
      A     "A1.7";
      AN    "E1.3";
      );
      =     "A1.0";
NETWORK
TITLE =
      A     "M11.2";
      A     "M32.2";
      O;
      A     "AUT";
      A     "M52.4";
      =     "A1.1";
NETWORK
TITLE =
      A     "On";
      =     L 0.0;
      A     L 0.0;
      A     DB21.DBX 476.0;
      =     M 2.1;
      A     L 0.0;
      A     DB21.DBX 476.1;
      =     M 2.1;
      A     L 0.0;
      A     DB21.DBX 476.2;
      =     M 2.1;
      A     L 0.0;
      A     DB21.DBX 476.3;
      =     M 2.1;
      A     L 0.0;
      A     DB21.DBX 476.4;
      =     M 2.1;
NETWORK
TITLE =
      A     "On";
      =     L 0.0;
      A     L 0.0;
      BLD   102;
      =     M 2.1;
      A     L 0.0;
      A     "ChangeFunc";
      =     M 2.1;
NETWORK
TITLE =
      A     "On";
      =     M 2.1;
END_FUNCTION

FUNCTION "FC19 - REPOSITIONING" : VOID	// FC 19
VERSION : 0.1
BEGIN
// (block stored without names or comments; labels and parameter names are numbered)
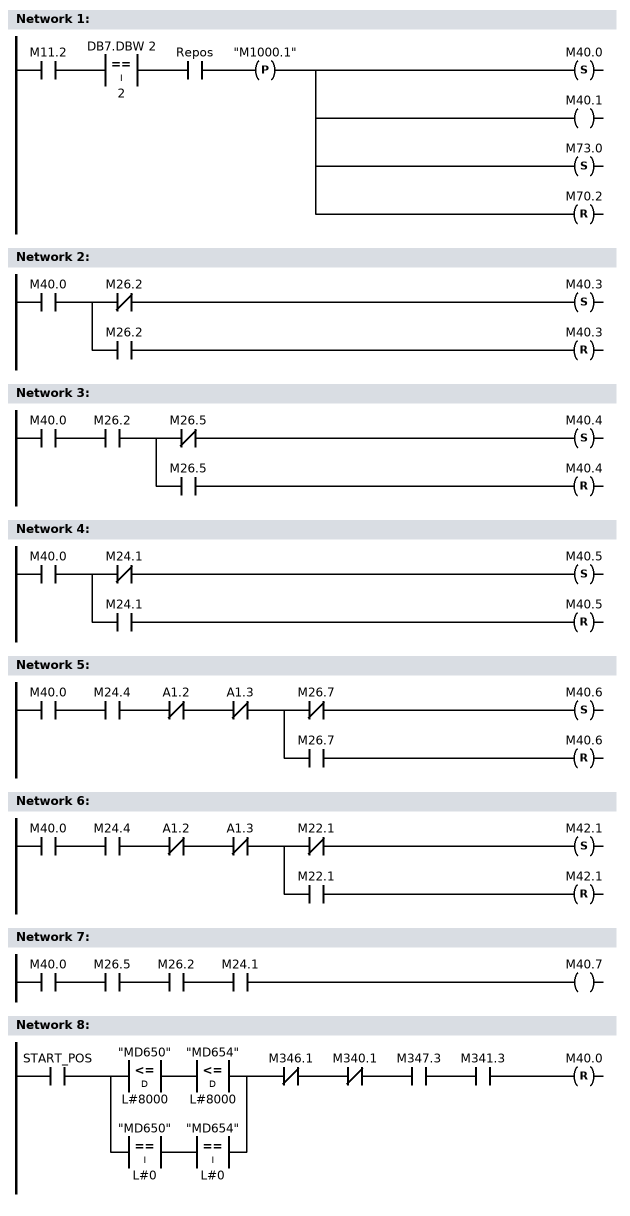
NETWORK
TITLE =
      A     "M11.2";
      A(;
      L     DB7.DBW 2;
      L     2;
      ==I;
      );
      A     "Repos";
      FP    "M1000.1";
      S     "M40.0";
      =     "M40.1";
      S     "M73.0";
      R     "M70.2";
NETWORK
TITLE =
      A     "M40.0";
      =     L 0.0;
      A     L 0.0;
      AN    "M26.2";
      S     "M40.3";
      A     L 0.0;
      A     "M26.2";
      R     "M40.3";
NETWORK
TITLE =
      A     "M40.0";
      A     "M26.2";
      =     L 0.0;
      A     L 0.0;
      AN    "M26.5";
      S     "M40.4";
      A     L 0.0;
      A     "M26.5";
      R     "M40.4";
NETWORK
TITLE =
      A     "M40.0";
      =     L 0.0;
      A     L 0.0;
      AN    "M24.1";
      S     "M40.5";
      A     L 0.0;
      A     "M24.1";
      R     "M40.5";
NETWORK
TITLE =
      A     "M40.0";
      A     "M24.4";
      AN    "A1.2";
      AN    "A1.3";
      =     L 0.0;
      A     L 0.0;
      AN    "M26.7";
      S     "M40.6";
      A     L 0.0;
      A     "M26.7";
      R     "M40.6";
NETWORK
TITLE =
      A     "M40.0";
      A     "M24.4";
      AN    "A1.2";
      AN    "A1.3";
      =     L 0.0;
      A     L 0.0;
      AN    "M22.1";
      S     "M42.1";
      A     L 0.0;
      A     "M22.1";
      R     "M42.1";
NETWORK
TITLE =
      A     "M40.0";
      A     "M26.5";
      A     "M26.2";
      A     "M24.1";
      =     "M40.7";
NETWORK
TITLE =
      A     "START_POS";
      A(;
      A(;
      L     "MD650";
      L     L#8000;
      <=D;
      );
      A(;
      L     "MD654";
      L     L#8000;
      <=D;
      );
      O;
      A(;
      L     "MD650";
      L     L#0;
      ==I;
      );
      A(;
      L     "MD654";
      L     L#0;
      ==I;
      );
      );
      AN    "M346.1";
      AN    "M340.1";
      A     "M347.3";
      A     "M341.3";
      R     "M40.0";
NETWORK
TITLE =
END_FUNCTION

FUNCTION "FC - AUTOMATIC" : VOID	// FC 24
VERSION : 0.1
BEGIN
// (block stored without names or comments; labels and parameter names are numbered)
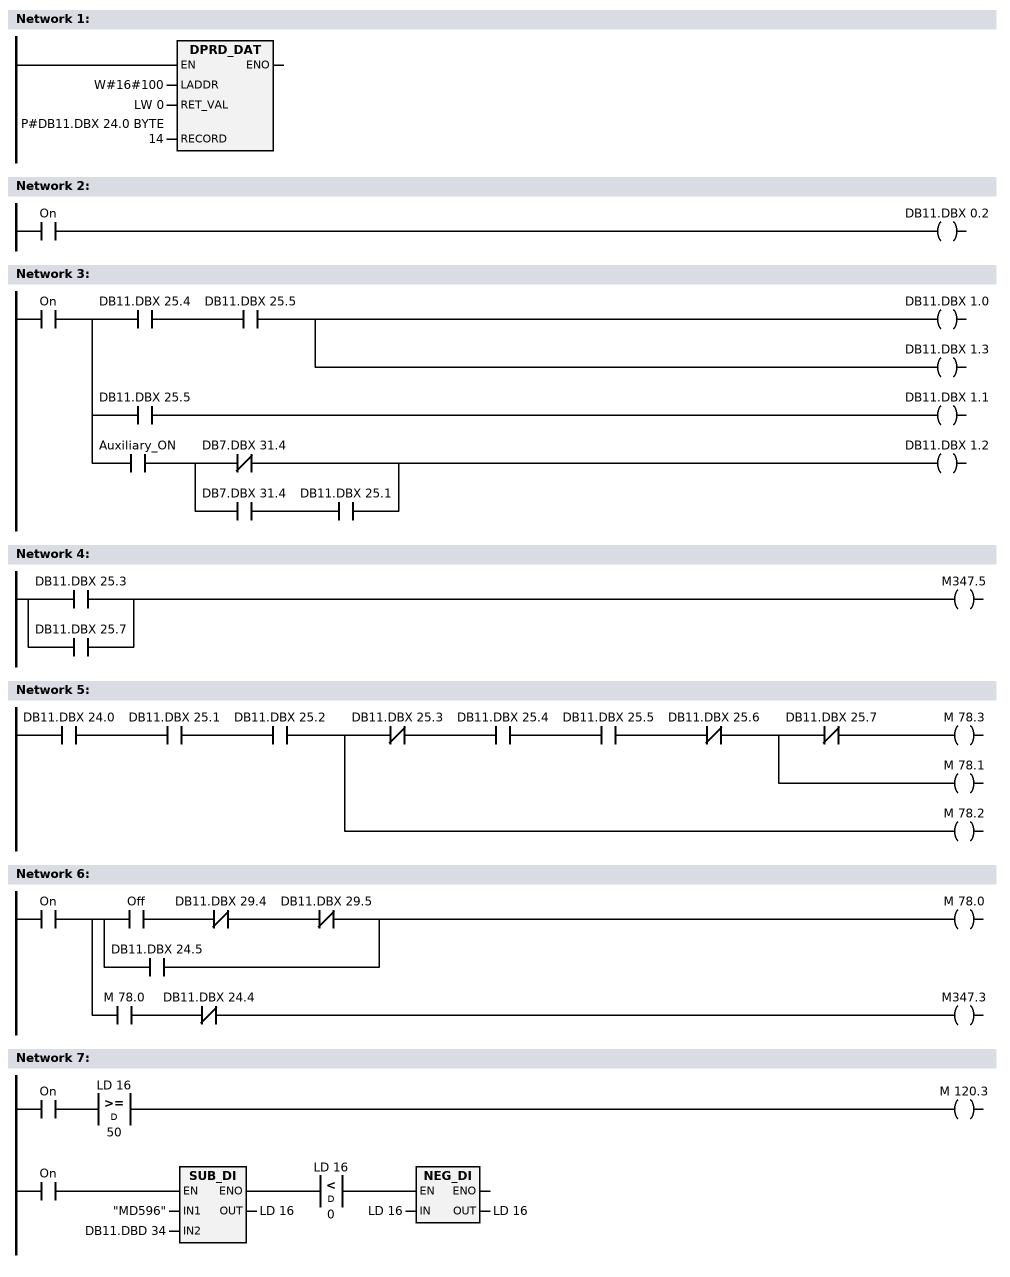
NETWORK
TITLE =
      CALL  "DPRD_DAT" (
           LADDR                    := W#16#100,
           RET_VAL                  := LW 0,
           RECORD                   := P#DB11.DBX 24.0 BYTE 14);
      NOP   0;
NETWORK
TITLE =
      A     "On";
      =     DB11.DBX 0.2;
NETWORK
TITLE =
      A     "On";
      =     L 20.0;
      A     L 20.0;
      A     DB11.DBX 25.4;
      A     DB11.DBX 25.5;
      =     DB11.DBX 1.0;
      =     DB11.DBX 1.3;
      A     L 20.0;
      A     DB11.DBX 25.5;
      =     DB11.DBX 1.1;
      A     L 20.0;
      A     "Auxiliary_ON";
      A(;
      ON    DB7.DBX 31.4;
      O;
      A     DB7.DBX 31.4;
      A     DB11.DBX 25.1;
      );
      =     DB11.DBX 1.2;
NETWORK
TITLE =
      O     DB11.DBX 25.3;
      O     DB11.DBX 25.7;
      =     "M347.5";
NETWORK
TITLE =
      A     DB11.DBX 24.0;
      A     DB11.DBX 25.1;
      A     DB11.DBX 25.2;
      =     L 20.0;
      A     L 20.0;
      AN    DB11.DBX 25.3;
      A     DB11.DBX 25.4;
      A     DB11.DBX 25.5;
      AN    DB11.DBX 25.6;
      =     L 20.1;
      A     L 20.1;
      AN    DB11.DBX 25.7;
      =     M 78.3;
      A     L 20.1;
      BLD   102;
      =     M 78.1;
      A     L 20.0;
      BLD   102;
      =     M 78.2;
NETWORK
TITLE =
      A     "On";
      =     L 20.0;
      A     L 20.0;
      A(;
      A     "Off";
      AN    DB11.DBX 29.4;
      AN    DB11.DBX 29.5;
      O     DB11.DBX 24.5;
      );
      =     M 78.0;
      A     L 20.0;
      A     M 78.0;
      AN    DB11.DBX 24.4;
      =     "M347.3";
NETWORK
TITLE =
      A     "On";
      =     L 20.0;
      A(;
      A     L 20.0;
      JNB   M001;
      L     "MD596";
      L     DB11.DBD 34;
      -D;
      T     LD 16;
      AN    OV;
      SAVE;
      CLR;
M001: A     BR;
      );
      A(;
      L     LD 16;
      L     0;
      <D;
      );
      JNB   M002;
      L     LD 16;
      NEGD;
      T     LD 16;
M002: NOP   0;
      A     L 20.0;
      A(;
      L     LD 16;
      L     50;
      >=D;
      );
      =     M 120.3;
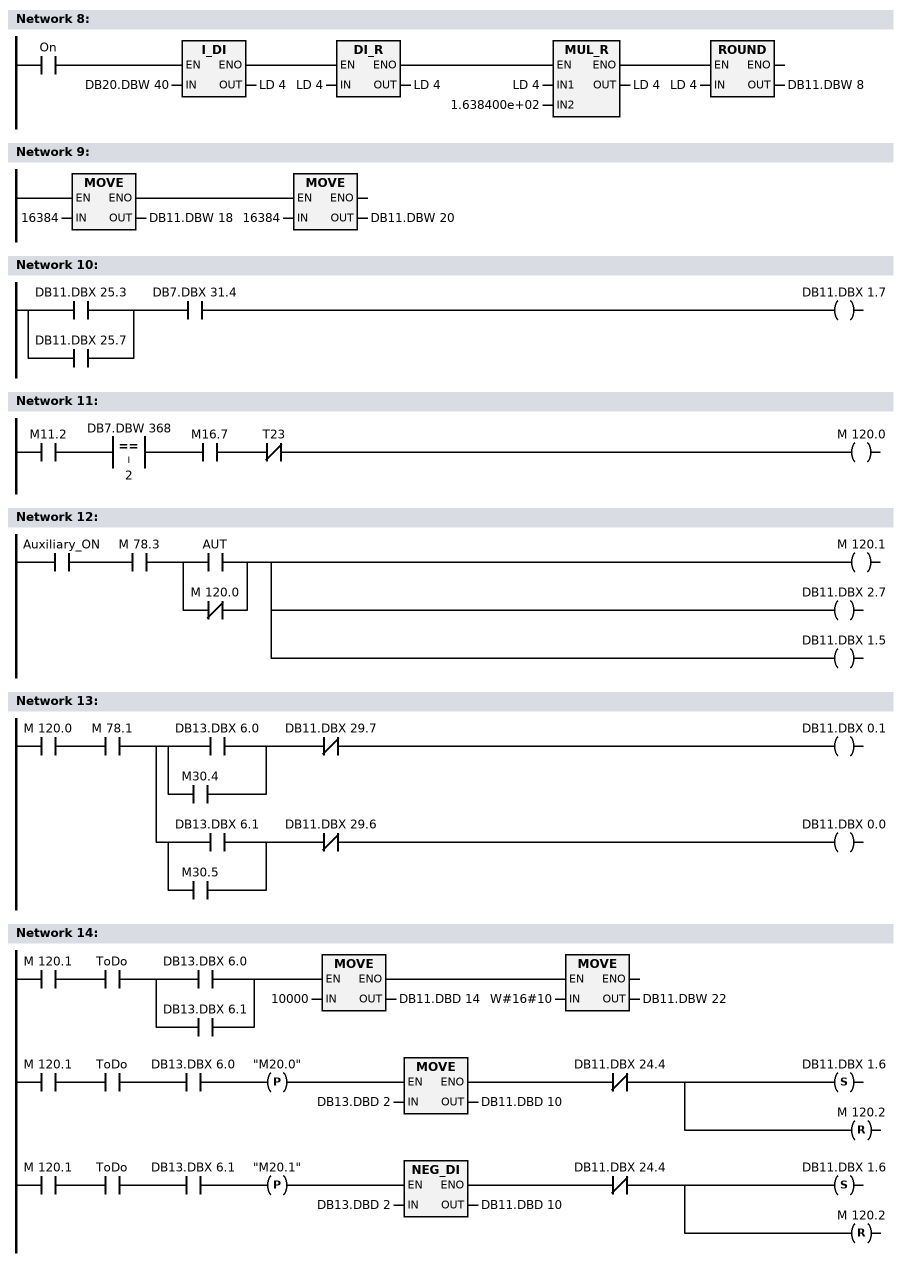
NETWORK
TITLE =
      A(;
      A(;
      A(;
      A     "On";
      JNB   M003;
      L     DB20.DBW 40;
      ITD;
      T     LD 4;
      SET;
      SAVE;
      CLR;
M003: A     BR;
      );
      JNB   M004;
      L     LD 4;
      DTR;
      T     LD 4;
      SET;
      SAVE;
      CLR;
M004: A     BR;
      );
      JNB   M005;
      L     LD 4;
      L     1.638400e+02;
      *R;
      T     LD 4;
      AN    OV;
      SAVE;
      CLR;
M005: A     BR;
      );
      JNB   M006;
      L     LD 4;
      RND;
      T     DB11.DBW 8;
M006: NOP   0;
NETWORK
TITLE =
      A(;
      L     16384;
      T     DB11.DBW 18;
      SET;
      SAVE;
      CLR;
      A     BR;
      );
      JNB   M007;
      L     16384;
      T     DB11.DBW 20;
M007: NOP   0;
NETWORK
TITLE =
      A(;
      O     DB11.DBX 25.3;
      O     DB11.DBX 25.7;
      );
      A     DB7.DBX 31.4;
      =     DB11.DBX 1.7;
NETWORK
TITLE =
      A     "M11.2";
      A(;
      L     DB7.DBW 368;
      L     2;
      ==I;
      );
      A     "M16.7";
      AN    "T23";
      =     M 120.0;
NETWORK
TITLE =
      A     "Auxiliary_ON";
      A     M 78.3;
      A(;
      O     "AUT";
      ON    M 120.0;
      );
      =     M 120.1;
      =     DB11.DBX 2.7;
      =     DB11.DBX 1.5;
NETWORK
TITLE =
      A     M 120.0;
      A     M 78.1;
      =     L 20.0;
      A     L 20.0;
      A(;
      O     DB13.DBX 6.0;
      O     "M30.4";
      );
      AN    DB11.DBX 29.7;
      =     DB11.DBX 0.1;
      A     L 20.0;
      A(;
      O     DB13.DBX 6.1;
      O     "M30.5";
      );
      AN    DB11.DBX 29.6;
      =     DB11.DBX 0.0;
NETWORK
TITLE =
      A     M 120.1;
      A     "ToDo";
      =     L 20.0;
      A(;
      A     L 20.0;
      A(;
      O     DB13.DBX 6.0;
      O     DB13.DBX 6.1;
      );
      JNB   M008;
      L     10000;
      T     DB11.DBD 14;
      SET;
      SAVE;
      CLR;
M008: A     BR;
      );
      JNB   M009;
      L     W#16#10;
      T     DB11.DBW 22;
M009: NOP   0;
      A(;
      A     L 20.0;
      A     DB13.DBX 6.0;
      FP    "M20.0";
      JNB   M010;
      L     DB13.DBD 2;
      T     DB11.DBD 10;
      SET;
      SAVE;
      CLR;
M010: A     BR;
      );
      AN    DB11.DBX 24.4;
      S     DB11.DBX 1.6;
      R     M 120.2;
      A(;
      A     L 20.0;
      A     DB13.DBX 6.1;
      FP    "M20.1";
      JNB   M011;
      L     DB13.DBD 2;
      NEGD;
      T     DB11.DBD 10;
      AN    OV;
      SAVE;
      CLR;
M011: A     BR;
      );
      AN    DB11.DBX 24.4;
      S     DB11.DBX 1.6;
      R     M 120.2;
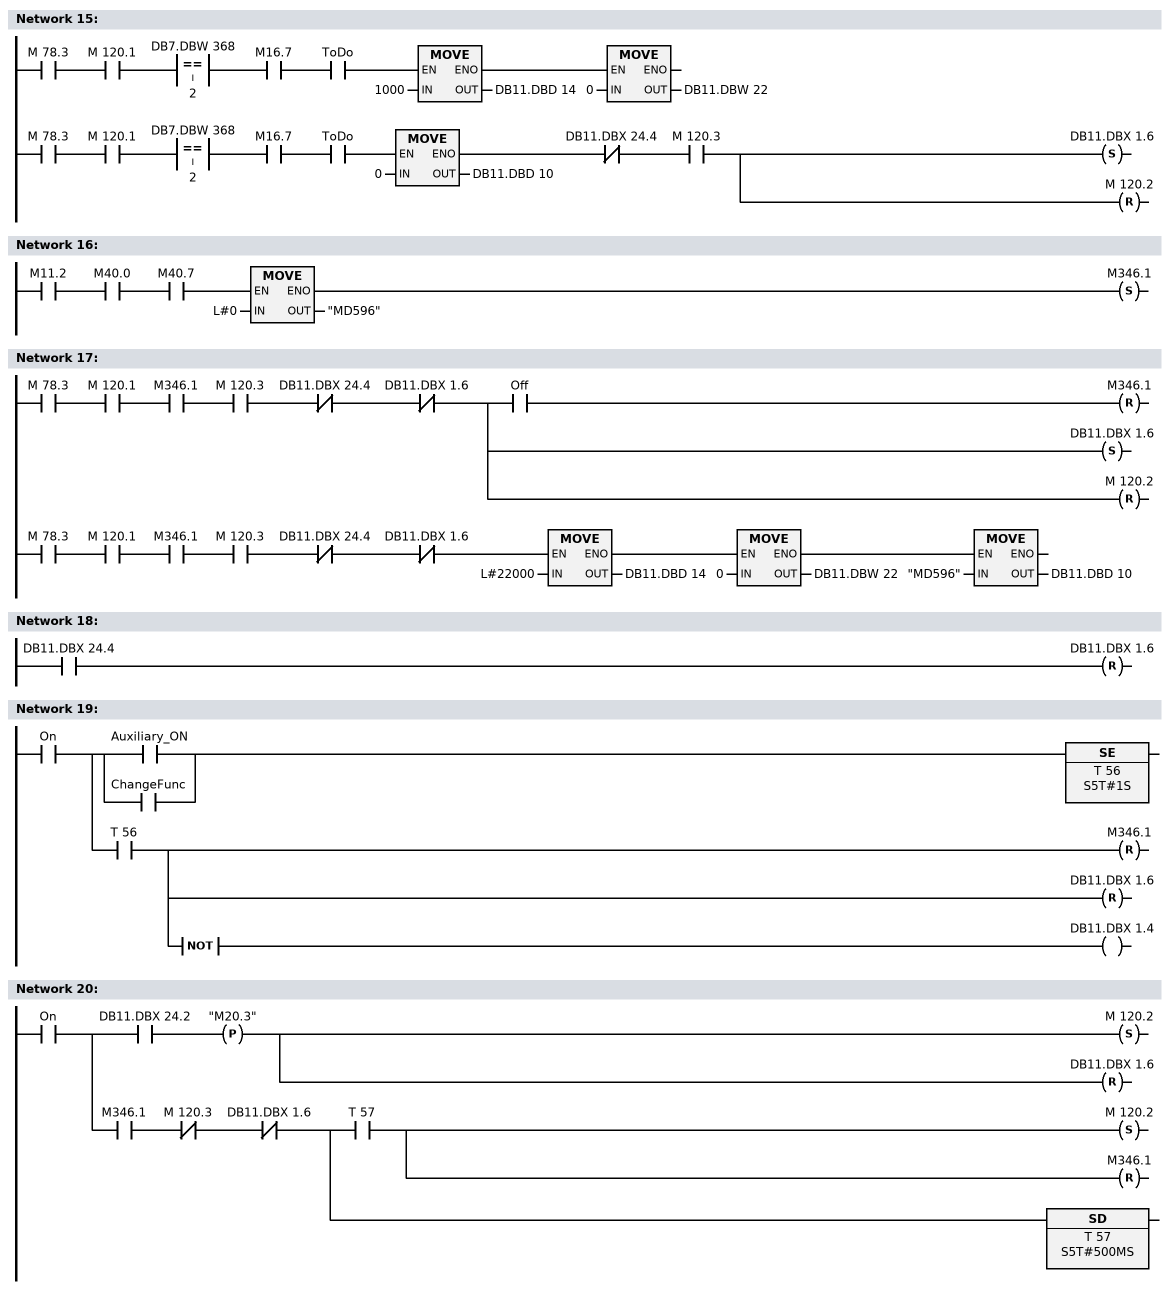
NETWORK
TITLE =
      A     M 78.3;
      A     M 120.1;
      A(;
      L     DB7.DBW 368;
      L     2;
      ==I;
      );
      A     "M16.7";
      =     L 20.0;
      A(;
      A     L 20.0;
      A     "ToDo";
      JNB   M012;
      L     1000;
      T     DB11.DBD 14;
      SET;
      SAVE;
      CLR;
M012: A     BR;
      );
      JNB   M013;
      L     0;
      T     DB11.DBW 22;
M013: NOP   0;
      A(;
      A     L 20.0;
      A     "ToDo";
      JNB   M014;
      L     0;
      T     DB11.DBD 10;
      SET;
      SAVE;
      CLR;
M014: A     BR;
      );
      AN    DB11.DBX 24.4;
      A     M 120.3;
      S     DB11.DBX 1.6;
      R     M 120.2;
NETWORK
TITLE =
      A     "M11.2";
      A     "M40.0";
      A     "M40.7";
      JNB   M015;
      L     L#0;
      T     "MD596";
      SET;
      SAVE;
      CLR;
M015: A     BR;
      S     "M346.1";
NETWORK
TITLE =
      A     M 78.3;
      A     M 120.1;
      A     "M346.1";
      A     M 120.3;
      AN    DB11.DBX 24.4;
      AN    DB11.DBX 1.6;
      =     L 20.0;
      A(;
      A(;
      A     L 20.0;
      JNB   M016;
      L     L#22000;
      T     DB11.DBD 14;
      SET;
      SAVE;
      CLR;
M016: A     BR;
      );
      JNB   M017;
      L     0;
      T     DB11.DBW 22;
      SET;
      SAVE;
      CLR;
M017: A     BR;
      );
      JNB   M018;
      L     "MD596";
      T     DB11.DBD 10;
M018: NOP   0;
      A     L 20.0;
      A     "Off";
      R     "M346.1";
      A     L 20.0;
      BLD   102;
      S     DB11.DBX 1.6;
      A     L 20.0;
      BLD   102;
      R     M 120.2;
NETWORK
TITLE =
      A     DB11.DBX 24.4;
      R     DB11.DBX 1.6;
NETWORK
TITLE =
      A     "On";
      =     L 20.0;
      A     L 20.0;
      A(;
      O     "Auxiliary_ON";
      O     "ChangeFunc";
      );
      L     S5T#1S;
      SE    T 56;
      A     L 20.0;
      A     T 56;
      =     L 20.1;
      A     L 20.1;
      BLD   102;
      R     "M346.1";
      A     L 20.1;
      BLD   102;
      R     DB11.DBX 1.6;
      A     L 20.1;
      NOT;
      =     DB11.DBX 1.4;
NETWORK
TITLE =
      A     "On";
      =     L 20.0;
      A     L 20.0;
      A     DB11.DBX 24.2;
      FP    "M20.3";
      S     M 120.2;
      R     DB11.DBX 1.6;
      A     L 20.0;
      A     "M346.1";
      AN    M 120.3;
      AN    DB11.DBX 1.6;
      =     L 20.1;
      A     L 20.1;
      A     T 57;
      S     M 120.2;
      R     "M346.1";
      A     L 20.1;
      BLD   102;
      L     S5T#500MS;
      SD    T 57;
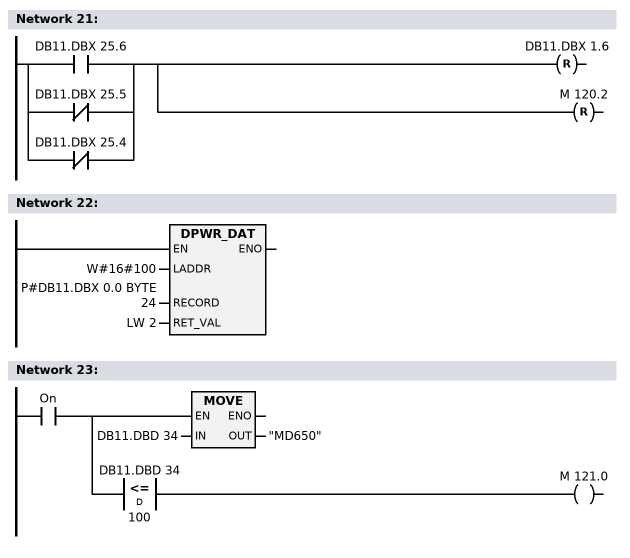
NETWORK
TITLE =
      O     DB11.DBX 25.6;
      ON    DB11.DBX 25.5;
      ON    DB11.DBX 25.4;
      R     DB11.DBX 1.6;
      R     M 120.2;
NETWORK
TITLE =
      CALL  "DPWR_DAT" (
           LADDR                    := W#16#100,
           RECORD                   := P#DB11.DBX 0.0 BYTE 24,
           RET_VAL                  := LW 2);
      NOP   0;
NETWORK
TITLE =
      A     "On";
      =     L 20.0;
      A     L 20.0;
      JNB   M019;
      L     DB11.DBD 34;
      T     "MD650";
M019: NOP   0;
      A     L 20.0;
      A(;
      L     DB11.DBD 34;
      L     100;
      <=D;
      );
      =     M 121.0;
END_FUNCTION

FUNCTION FC 25 : VOID
VERSION : 0.1
BEGIN
// (block stored without names or comments; labels and parameter names are numbered)
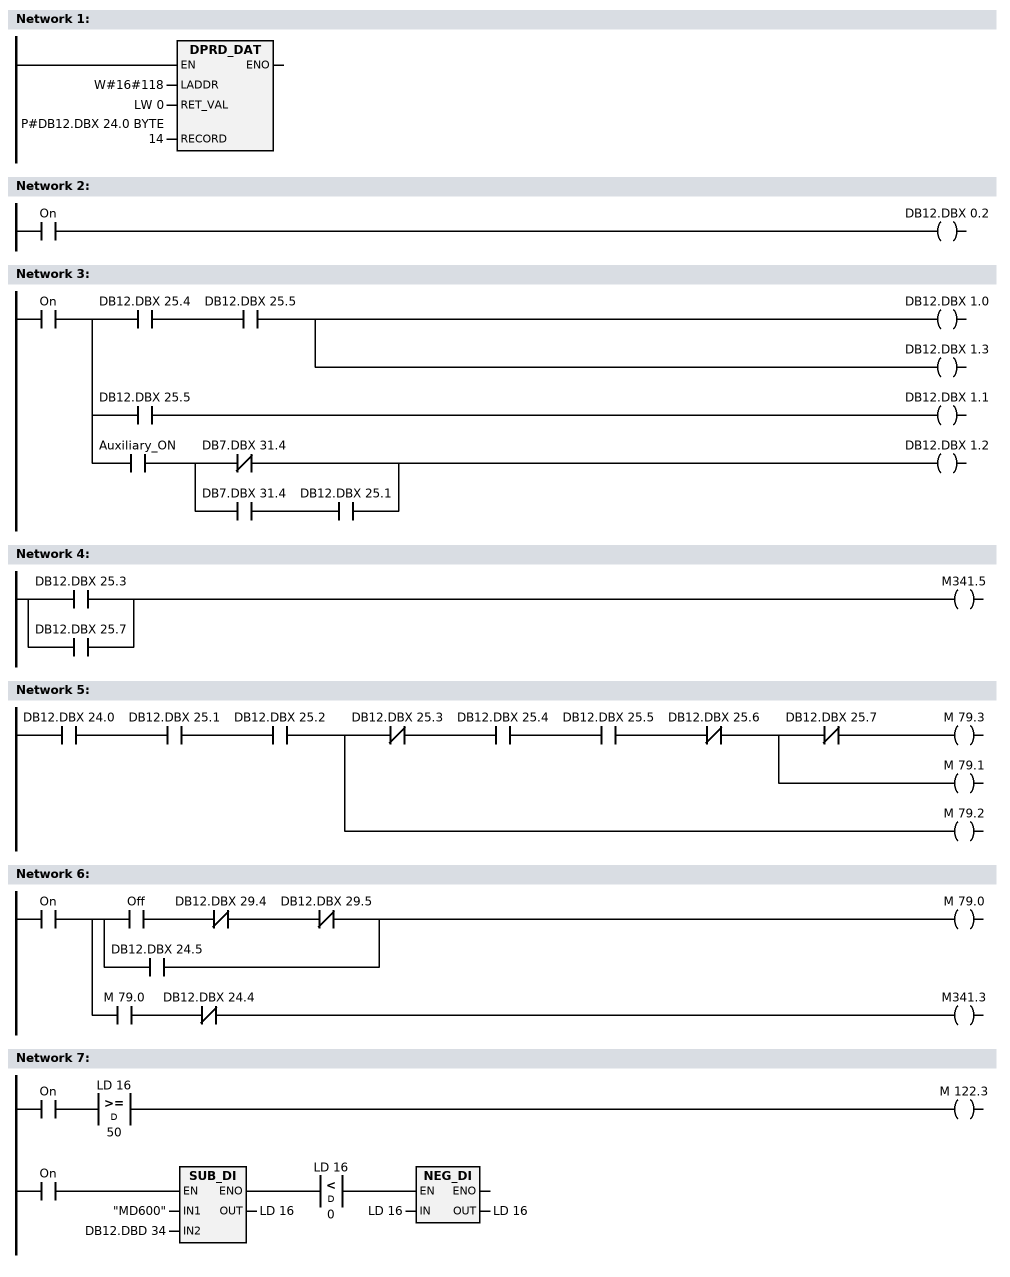
NETWORK
TITLE =
      CALL  "DPRD_DAT" (
           LADDR                    := W#16#118,
           RET_VAL                  := LW 0,
           RECORD                   := P#DB12.DBX 24.0 BYTE 14);
      NOP   0;
NETWORK
TITLE =
      A     "On";
      =     DB12.DBX 0.2;
NETWORK
TITLE =
      A     "On";
      =     L 20.0;
      A     L 20.0;
      A     DB12.DBX 25.4;
      A     DB12.DBX 25.5;
      =     DB12.DBX 1.0;
      =     DB12.DBX 1.3;
      A     L 20.0;
      A     DB12.DBX 25.5;
      =     DB12.DBX 1.1;
      A     L 20.0;
      A     "Auxiliary_ON";
      A(;
      ON    DB7.DBX 31.4;
      O;
      A     DB7.DBX 31.4;
      A     DB12.DBX 25.1;
      );
      =     DB12.DBX 1.2;
NETWORK
TITLE =
      O     DB12.DBX 25.3;
      O     DB12.DBX 25.7;
      =     "M341.5";
NETWORK
TITLE =
      A     DB12.DBX 24.0;
      A     DB12.DBX 25.1;
      A     DB12.DBX 25.2;
      =     L 20.0;
      A     L 20.0;
      AN    DB12.DBX 25.3;
      A     DB12.DBX 25.4;
      A     DB12.DBX 25.5;
      AN    DB12.DBX 25.6;
      =     L 20.1;
      A     L 20.1;
      AN    DB12.DBX 25.7;
      =     M 79.3;
      A     L 20.1;
      BLD   102;
      =     M 79.1;
      A     L 20.0;
      BLD   102;
      =     M 79.2;
NETWORK
TITLE =
      A     "On";
      =     L 20.0;
      A     L 20.0;
      A(;
      A     "Off";
      AN    DB12.DBX 29.4;
      AN    DB12.DBX 29.5;
      O     DB12.DBX 24.5;
      );
      =     M 79.0;
      A     L 20.0;
      A     M 79.0;
      AN    DB12.DBX 24.4;
      =     "M341.3";
NETWORK
TITLE =
      A     "On";
      =     L 20.0;
      A(;
      A     L 20.0;
      JNB   M001;
      L     "MD600";
      L     DB12.DBD 34;
      -D;
      T     LD 16;
      AN    OV;
      SAVE;
      CLR;
M001: A     BR;
      );
      A(;
      L     LD 16;
      L     0;
      <D;
      );
      JNB   M002;
      L     LD 16;
      NEGD;
      T     LD 16;
M002: NOP   0;
      A     L 20.0;
      A(;
      L     LD 16;
      L     50;
      >=D;
      );
      =     M 122.3;
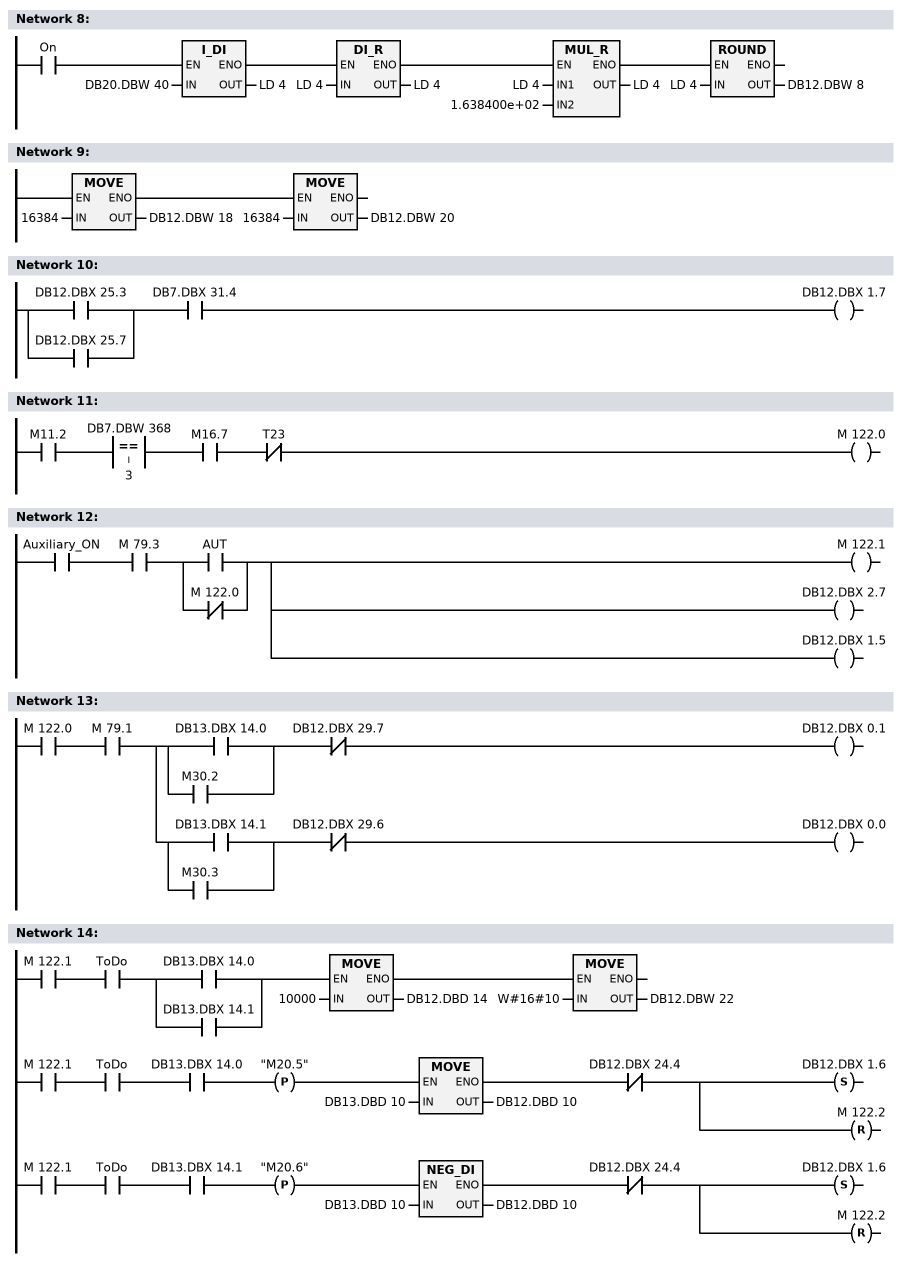
NETWORK
TITLE =
      A(;
      A(;
      A(;
      A     "On";
      JNB   M003;
      L     DB20.DBW 40;
      ITD;
      T     LD 4;
      SET;
      SAVE;
      CLR;
M003: A     BR;
      );
      JNB   M004;
      L     LD 4;
      DTR;
      T     LD 4;
      SET;
      SAVE;
      CLR;
M004: A     BR;
      );
      JNB   M005;
      L     LD 4;
      L     1.638400e+02;
      *R;
      T     LD 4;
      AN    OV;
      SAVE;
      CLR;
M005: A     BR;
      );
      JNB   M006;
      L     LD 4;
      RND;
      T     DB12.DBW 8;
M006: NOP   0;
NETWORK
TITLE =
      A(;
      L     16384;
      T     DB12.DBW 18;
      SET;
      SAVE;
      CLR;
      A     BR;
      );
      JNB   M007;
      L     16384;
      T     DB12.DBW 20;
M007: NOP   0;
NETWORK
TITLE =
      A(;
      O     DB12.DBX 25.3;
      O     DB12.DBX 25.7;
      );
      A     DB7.DBX 31.4;
      =     DB12.DBX 1.7;
NETWORK
TITLE =
      A     "M11.2";
      A(;
      L     DB7.DBW 368;
      L     3;
      ==I;
      );
      A     "M16.7";
      AN    "T23";
      =     M 122.0;
NETWORK
TITLE =
      A     "Auxiliary_ON";
      A     M 79.3;
      A(;
      O     "AUT";
      ON    M 122.0;
      );
      =     M 122.1;
      =     DB12.DBX 2.7;
      =     DB12.DBX 1.5;
NETWORK
TITLE =
      A     M 122.0;
      A     M 79.1;
      =     L 20.0;
      A     L 20.0;
      A(;
      O     DB13.DBX 14.0;
      O     "M30.2";
      );
      AN    DB12.DBX 29.7;
      =     DB12.DBX 0.1;
      A     L 20.0;
      A(;
      O     DB13.DBX 14.1;
      O     "M30.3";
      );
      AN    DB12.DBX 29.6;
      =     DB12.DBX 0.0;
NETWORK
TITLE =
      A     M 122.1;
      A     "ToDo";
      =     L 20.0;
      A(;
      A     L 20.0;
      A(;
      O     DB13.DBX 14.0;
      O     DB13.DBX 14.1;
      );
      JNB   M008;
      L     10000;
      T     DB12.DBD 14;
      SET;
      SAVE;
      CLR;
M008: A     BR;
      );
      JNB   M009;
      L     W#16#10;
      T     DB12.DBW 22;
M009: NOP   0;
      A(;
      A     L 20.0;
      A     DB13.DBX 14.0;
      FP    "M20.5";
      JNB   M010;
      L     DB13.DBD 10;
      T     DB12.DBD 10;
      SET;
      SAVE;
      CLR;
M010: A     BR;
      );
      AN    DB12.DBX 24.4;
      S     DB12.DBX 1.6;
      R     M 122.2;
      A(;
      A     L 20.0;
      A     DB13.DBX 14.1;
      FP    "M20.6";
      JNB   M011;
      L     DB13.DBD 10;
      NEGD;
      T     DB12.DBD 10;
      AN    OV;
      SAVE;
      CLR;
M011: A     BR;
      );
      AN    DB12.DBX 24.4;
      S     DB12.DBX 1.6;
      R     M 122.2;
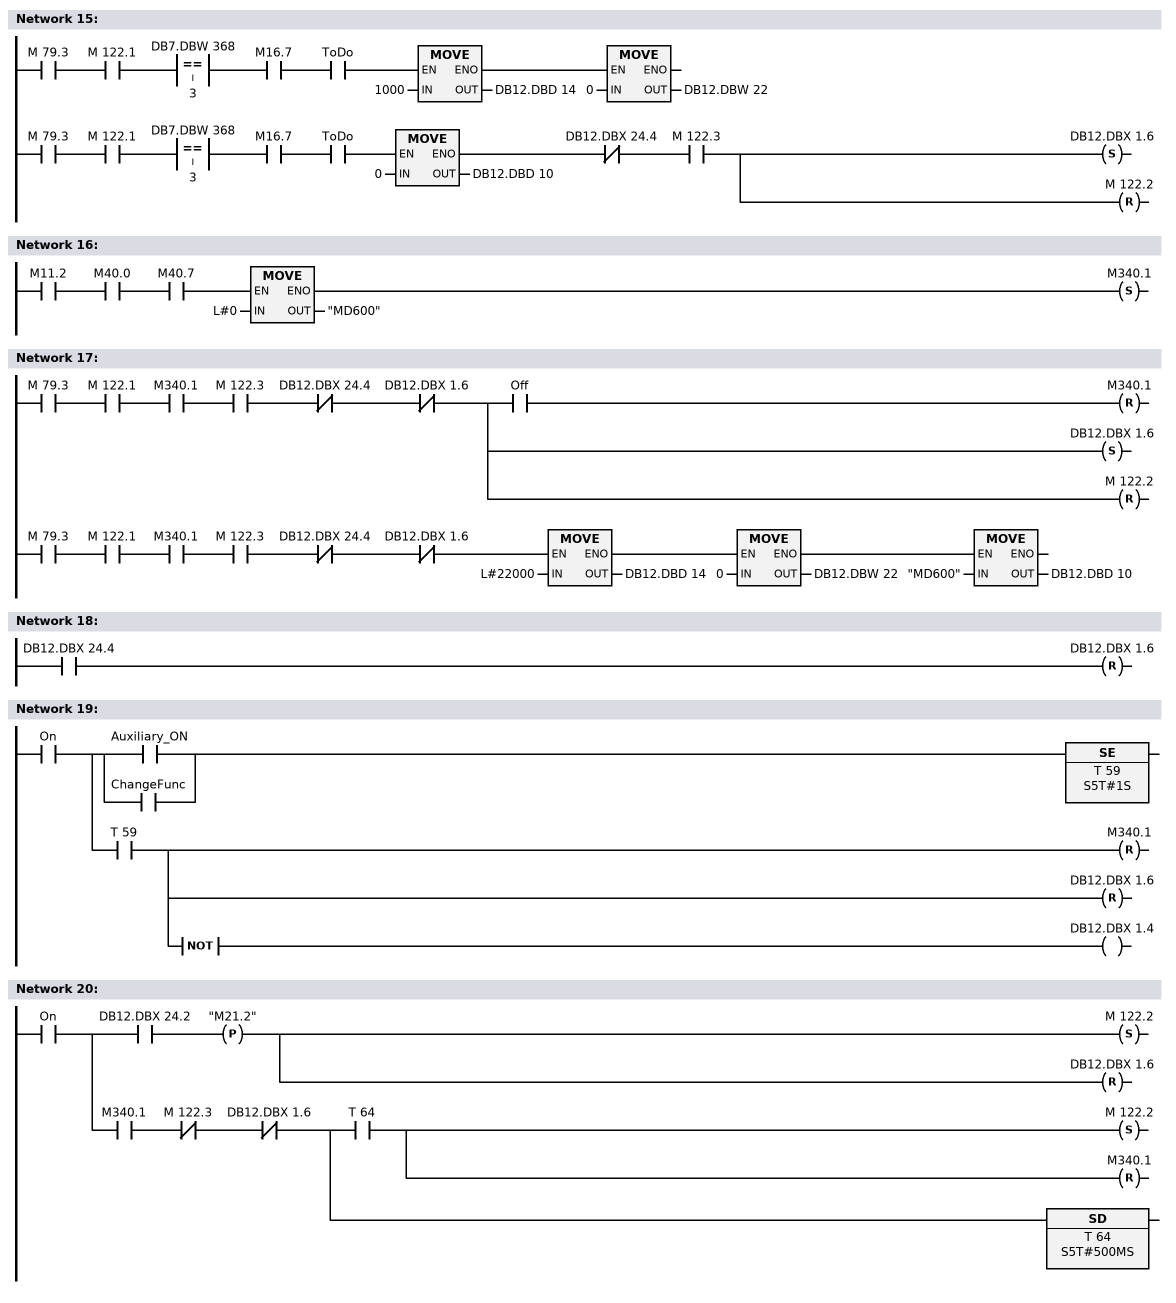
NETWORK
TITLE =
      A     M 79.3;
      A     M 122.1;
      A(;
      L     DB7.DBW 368;
      L     3;
      ==I;
      );
      A     "M16.7";
      =     L 20.0;
      A(;
      A     L 20.0;
      A     "ToDo";
      JNB   M012;
      L     1000;
      T     DB12.DBD 14;
      SET;
      SAVE;
      CLR;
M012: A     BR;
      );
      JNB   M013;
      L     0;
      T     DB12.DBW 22;
M013: NOP   0;
      A(;
      A     L 20.0;
      A     "ToDo";
      JNB   M014;
      L     0;
      T     DB12.DBD 10;
      SET;
      SAVE;
      CLR;
M014: A     BR;
      );
      AN    DB12.DBX 24.4;
      A     M 122.3;
      S     DB12.DBX 1.6;
      R     M 122.2;
NETWORK
TITLE =
      A     "M11.2";
      A     "M40.0";
      A     "M40.7";
      JNB   M015;
      L     L#0;
      T     "MD600";
      SET;
      SAVE;
      CLR;
M015: A     BR;
      S     "M340.1";
NETWORK
TITLE =
      A     M 79.3;
      A     M 122.1;
      A     "M340.1";
      A     M 122.3;
      AN    DB12.DBX 24.4;
      AN    DB12.DBX 1.6;
      =     L 20.0;
      A(;
      A(;
      A     L 20.0;
      JNB   M016;
      L     L#22000;
      T     DB12.DBD 14;
      SET;
      SAVE;
      CLR;
M016: A     BR;
      );
      JNB   M017;
      L     0;
      T     DB12.DBW 22;
      SET;
      SAVE;
      CLR;
M017: A     BR;
      );
      JNB   M018;
      L     "MD600";
      T     DB12.DBD 10;
M018: NOP   0;
      A     L 20.0;
      A     "Off";
      R     "M340.1";
      A     L 20.0;
      BLD   102;
      S     DB12.DBX 1.6;
      A     L 20.0;
      BLD   102;
      R     M 122.2;
NETWORK
TITLE =
      A     DB12.DBX 24.4;
      R     DB12.DBX 1.6;
NETWORK
TITLE =
      A     "On";
      =     L 20.0;
      A     L 20.0;
      A(;
      O     "Auxiliary_ON";
      O     "ChangeFunc";
      );
      L     S5T#1S;
      SE    T 59;
      A     L 20.0;
      A     T 59;
      =     L 20.1;
      A     L 20.1;
      BLD   102;
      R     "M340.1";
      A     L 20.1;
      BLD   102;
      R     DB12.DBX 1.6;
      A     L 20.1;
      NOT;
      =     DB12.DBX 1.4;
NETWORK
TITLE =
      A     "On";
      =     L 20.0;
      A     L 20.0;
      A     DB12.DBX 24.2;
      FP    "M21.2";
      S     M 122.2;
      R     DB12.DBX 1.6;
      A     L 20.0;
      A     "M340.1";
      AN    M 122.3;
      AN    DB12.DBX 1.6;
      =     L 20.1;
      A     L 20.1;
      A     T 64;
      S     M 122.2;
      R     "M340.1";
      A     L 20.1;
      BLD   102;
      L     S5T#500MS;
      SD    T 64;
